// TwinCAT 3 PLC project plc_lfe_vac
// ProgramVersion: 3.1.4022.3
// libraries:
//   L2SI Vacuum Library-TEST, * (SLAC)
//   LCLS General, * (SLAC)
//   PMPS, * (SLAC - LCLS)
//   Tc2_Standard, * (Beckhoff Automation GmbH)
//   Tc2_System, * (Beckhoff Automation GmbH)
//   Tc3_Module, * (Beckhoff Automation GmbH)
// project tree:
//   GVLs/ GVL_Devices.TcGVL, GVL_PMPS.TcGVL (not stored), GVL_PLC_Interfaces.TcGVL (not stored), GVL_Variables.TcGVL
//   / PlcTask.TcTTO (not stored)
//   POUs/ DIAGNOSTICS.TcPOU, MAIN.TcPOU
// real-time tasks:
//   TASK PlcTask: cycle T#10ms, priority 20, ADS port 350
// I/O:
//   DEVICE Device 1 (EtherCAT), AmsNetId 172.21.88.138.2.1
//     PLC_E0_EK1200
// variable links:
//   plc_lfe_vac/plc_lfe_vac Instance <-> Device 1 (EtherCAT)/PLC_E0_EK1200/PLC_E11_EK1122_FEE_Stands/FEE_L0S10_EP1_EP2338-0002
//     PlcTask Inputs/GVL_Devices.MR1L0_HOMS_VGC_01.i_xClsLS <-> Channel 2/Input
//     PlcTask Inputs/GVL_Devices.MR1L0_HOMS_VGC_01.i_xOpnLS <-> Channel 1/Input
//     PlcTask Outputs/GVL_Devices.MR1L0_HOMS_VGC_01.q_xOPN_DO <-> Channel 11/Output
//   plc_lfe_vac/plc_lfe_vac Instance <-> Device 1 (EtherCAT)/PLC_E0_EK1200/PLC_E11_EK1122_FEE_Stands/FEE_L0S14_EP1_EP2338-0002
//     PlcTask Inputs/GVL_Devices.BT2L0_PLEG_VGC_01.i_xClsLS <-> Channel 2/Input
//     PlcTask Inputs/GVL_Devices.BT2L0_PLEG_VGC_01.i_xOpnLS <-> Channel 1/Input
//     PlcTask Outputs/GVL_Devices.BT2L0_PLEG_VGC_01.q_xOPN_DO <-> Channel 11/Output
//   plc_lfe_vac/plc_lfe_vac Instance <-> Device 1 (EtherCAT)/PLC_E0_EK1200/PLC_E11_EK1122_FEE_Stands/FEE_L0S14_EP2_EP3174-0002
//     PlcTask Inputs/GVL_Devices.BT2L0_PLEG_GCC_01.i_iPRESS_R <-> AI Standard Channel 4/Value
//     PlcTask Inputs/GVL_Devices.BT2L0_PLEG_GPI_01.i_iPRESS_R <-> AI Standard Channel 3/Value
//     PlcTask Inputs/GVL_Devices.MR1L1_TXI_GCC_01.i_iPRESS_R <-> AI Standard Channel 2/Value
//     PlcTask Inputs/GVL_Devices.MR1L1_TXI_GPI_01.i_iPRESS_R <-> AI Standard Channel 1/Value
//   plc_lfe_vac/plc_lfe_vac Instance <-> Device 1 (EtherCAT)/PLC_E0_EK1200/PLC_E11_EK1122_FEE_Stands/FEE_L0S14_EP3_EP2624-0002
//     PlcTask Outputs/GVL_Devices.BT2L0_PLEG_GCC_01.q_xHV_DIS <-> Channel 4/Output
//     PlcTask Outputs/GVL_Devices.MR1L1_TXI_GCC_01.q_xHV_DIS <-> Channel 2/Output
//   plc_lfe_vac/plc_lfe_vac Instance <-> Device 1 (EtherCAT)/PLC_E0_EK1200/PLC_E11_EK1122_FEE_Stands/FEE_L0S18_EP1_EP2338-0002
//     PlcTask Inputs/GVL_Devices.MR2L0_HOMS_VGC_01.i_xClsLS <-> Channel 2/Input
//     PlcTask Inputs/GVL_Devices.MR2L0_HOMS_VGC_01.i_xOpnLS <-> Channel 1/Input
//     PlcTask Inputs/GVL_Devices.TV1L1_VGC_01.i_xClsLS <-> Channel 6/Input
//     PlcTask Inputs/GVL_Devices.TV1L1_VGC_01.i_xOpnLS <-> Channel 5/Input
//     PlcTask Outputs/GVL_Devices.MR2L0_HOMS_VGC_01.q_xOPN_DO <-> Channel 11/Output
//     PlcTask Outputs/GVL_Devices.TV1L1_VGC_01.q_xOPN_DO <-> Channel 15/Output
//   plc_lfe_vac/plc_lfe_vac Instance <-> Device 1 (EtherCAT)/PLC_E0_EK1200/PLC_E11_EK1122_FEE_Stands/FEE_L0S18_EP2_EP3174-0002
//     PlcTask Inputs/GVL_Devices.MR2L0_HOMS_GCC_01.i_iPRESS_R <-> AI Standard Channel 2/Value
//     PlcTask Inputs/GVL_Devices.MR2L0_HOMS_GPI_01.i_iPRESS_R <-> AI Standard Channel 1/Value
//   plc_lfe_vac/plc_lfe_vac Instance <-> Device 1 (EtherCAT)/PLC_E0_EK1200/PLC_E11_EK1122_FEE_Stands/FEE_L0S18_EP3_EP2624-0002
//     PlcTask Outputs/GVL_Devices.MR2L0_HOMS_GCC_01.q_xHV_DIS <-> Channel 2/Output
//   plc_lfe_vac/plc_lfe_vac Instance <-> Device 1 (EtherCAT)/PLC_E0_EK1200/PLC_E11_EK1122_FEE_Stands/FEE_L0S19_EP1_EP2338-0002
//     PlcTask Inputs/GVL_Devices.MR2L0_HOMS_VGC_02.i_xClsLS <-> Channel 2/Input
//     PlcTask Inputs/GVL_Devices.MR2L0_HOMS_VGC_02.i_xOpnLS <-> Channel 1/Input
//     PlcTask Inputs/GVL_Devices.PC2L1_L2SI_VGC_01.i_xClsLS <-> Channel 6/Input
//     PlcTask Inputs/GVL_Devices.PC2L1_L2SI_VGC_01.i_xOpnLS <-> Channel 5/Input
//     PlcTask Outputs/GVL_Devices.MR2L0_HOMS_VGC_02.q_xOPN_DO <-> Channel 11/Output
//     PlcTask Outputs/GVL_Devices.PC2L1_L2SI_VGC_01.q_xOPN_DO <-> Channel 15/Output
//   plc_lfe_vac/plc_lfe_vac Instance <-> Device 1 (EtherCAT)/PLC_E0_EK1200/PLC_E11_EK1122_FEE_Stands/FEE_L0S21-2_EP1_EP3174-0002
//     PlcTask Inputs/GVL_Devices.ST1L0_XTES_GCC_01.i_iPRESS_R <-> AI Standard Channel 2/Value
//     PlcTask Inputs/GVL_Devices.ST1L0_XTES_GPI_01.i_iPRESS_R <-> AI Standard Channel 1/Value
//   plc_lfe_vac/plc_lfe_vac Instance <-> Device 1 (EtherCAT)/PLC_E0_EK1200/PLC_E11_EK1122_FEE_Stands/FEE_L0S21-2_EP2_EP2624-0002
//     PlcTask Outputs/GVL_Devices.ST1L0_XTES_GCC_01.q_xHV_DIS <-> Channel 2/Output
//   plc_lfe_vac/plc_lfe_vac Instance <-> Device 1 (EtherCAT)/PLC_E0_EK1200/PLC_E11_EK1122_FEE_Stands/FEE_L0S2_EP1_EP2338-0002
//     PlcTask Inputs/GVL_Devices.TV2L0_VGC_02.i_xClsLS <-> Channel 2/Input
//     PlcTask Inputs/GVL_Devices.TV2L0_VGC_02.i_xOpnLS <-> Channel 1/Input
//     PlcTask Outputs/GVL_Devices.TV2L0_VGC_02.q_xOPN_DO <-> Channel 11/Output
//   plc_lfe_vac/plc_lfe_vac Instance <-> Device 1 (EtherCAT)/PLC_E0_EK1200/PLC_E11_EK1122_FEE_Stands/FEE_L0S8_EP1_EP2338-0002
//     PlcTask Inputs/GVL_Devices.PC1L0_XTES_VGC_01.i_xClsLS <-> Channel 2/Input
//     PlcTask Inputs/GVL_Devices.PC1L0_XTES_VGC_01.i_xOpnLS <-> Channel 1/Input
//     PlcTask Outputs/GVL_Devices.PC1L0_XTES_VGC_01.q_xOPN_DO <-> Channel 11/Output
//   plc_lfe_vac/plc_lfe_vac Instance <-> Device 1 (EtherCAT)/PLC_E0_EK1200/PLC_E12_EK1122_H11_H12/H11_L0S2_EP1_EP2338-0002
//     PlcTask Inputs/GVL_Devices.TV4L0_VGC_01.i_xClsLS <-> Channel 2/Input
//     PlcTask Inputs/GVL_Devices.TV4L0_VGC_01.i_xOpnLS <-> Channel 1/Input
//     PlcTask Outputs/GVL_Devices.TV4L0_VGC_01.q_xOPN_DO <-> Channel 11/Output
//   plc_lfe_vac/plc_lfe_vac Instance <-> Device 1 (EtherCAT)/PLC_E0_EK1200/PLC_E12_EK1122_H11_H12/H11_L0S2_EP2_EP3174-0002
//     PlcTask Inputs/GVL_Devices.TV4L0_GCC_01.i_iPRESS_R <-> AI Standard Channel 2/Value
//     PlcTask Inputs/GVL_Devices.TV4L0_GPI_01.i_iPRESS_R <-> AI Standard Channel 1/Value
//   plc_lfe_vac/plc_lfe_vac Instance <-> Device 1 (EtherCAT)/PLC_E0_EK1200/PLC_E12_EK1122_H11_H12/H11_L0S2_EP3_EP2624-0002
//     PlcTask Outputs/GVL_Devices.TV4L0_GCC_01.q_xHV_DIS <-> Channel 2/Output
//   plc_lfe_vac/plc_lfe_vac Instance <-> Device 1 (EtherCAT)/PLC_E0_EK1200/PLC_E12_EK1122_H11_H12/H11_L0S9_EP1_EP3174-0002
//     PlcTask Inputs/GVL_Devices.TV4L0_GCC_02.i_iPRESS_R <-> AI Standard Channel 2/Value
//     PlcTask Inputs/GVL_Devices.TV4L0_GPI_02.i_iPRESS_R <-> AI Standard Channel 1/Value
//   plc_lfe_vac/plc_lfe_vac Instance <-> Device 1 (EtherCAT)/PLC_E0_EK1200/PLC_E12_EK1122_H11_H12/H11_L0S9_EP2_EP2624-0002
//     PlcTask Outputs/GVL_Devices.TV4L0_GCC_02.q_xHV_DIS <-> Channel 2/Output
//   plc_lfe_vac/plc_lfe_vac Instance <-> Device 1 (EtherCAT)/PLC_E0_EK1200/PLC_E12_EK1122_H11_H12/H12_L0S1_EP1_EP3174-0002
//     PlcTask Inputs/GVL_Devices.TV5L0_GCC_01.i_iPRESS_R <-> AI Standard Channel 2/Value
//     PlcTask Inputs/GVL_Devices.TV5L0_GPI_01.i_iPRESS_R <-> AI Standard Channel 1/Value
//   plc_lfe_vac/plc_lfe_vac Instance <-> Device 1 (EtherCAT)/PLC_E0_EK1200/PLC_E12_EK1122_H11_H12/H12_L0S1_EP2_EP2624-0002
//     PlcTask Outputs/GVL_Devices.TV5L0_GCC_01.q_xHV_DIS <-> Channel 2/Output
//   plc_lfe_vac/plc_lfe_vac Instance <-> Device 1 (EtherCAT)/PLC_E0_EK1200/PLC_E12_EK1122_H11_H12/H12_L0S3_EP1_EP2338-0002
//     PlcTask Inputs/GVL_Devices.TV5L0_VGC_01.i_xClsLS <-> Channel 2/Input
//     PlcTask Inputs/GVL_Devices.TV5L0_VGC_01.i_xOpnLS <-> Channel 1/Input
//     PlcTask Outputs/GVL_Devices.TV5L0_VGC_01.q_xOPN_DO <-> Channel 11/Output
//   plc_lfe_vac/plc_lfe_vac Instance <-> Device 1 (EtherCAT)/PLC_E0_EK1200/PLC_E12_EK1122_H11_H12/H12_L0S3_EP2_EP3174-0002
//     PlcTask Inputs/GVL_Devices.TV5L0_GCC_02.i_iPRESS_R <-> AI Standard Channel 2/Value
//     PlcTask Inputs/GVL_Devices.TV5L0_GCC_03.i_iPRESS_R <-> AI Standard Channel 4/Value
//     PlcTask Inputs/GVL_Devices.TV5L0_GPI_02.i_iPRESS_R <-> AI Standard Channel 1/Value
//   plc_lfe_vac/plc_lfe_vac Instance <-> Device 1 (EtherCAT)/PLC_E0_EK1200/PLC_E12_EK1122_H11_H12/H12_L0S3_EP3_EP2624-0002
//     PlcTask Outputs/GVL_Devices.TV5L0_GCC_02.q_xHV_DIS <-> Channel 2/Output
//     PlcTask Outputs/GVL_Devices.TV5L0_GCC_03.q_xHV_DIS <-> Channel 4/Output
//   plc_lfe_vac/plc_lfe_vac Instance <-> Device 1 (EtherCAT)/PLC_E0_EK1200/PLC_E12_EK1122_H11_H12/H12_L0S6_EP1_EP2338-0002
//     PlcTask Inputs/GVL_Devices.TV6L0_VGC_01.i_xClsLS <-> Channel 2/Input
//     PlcTask Inputs/GVL_Devices.TV6L0_VGC_01.i_xOpnLS <-> Channel 1/Input
//     PlcTask Outputs/GVL_Devices.TV6L0_VGC_01.q_xOPN_DO <-> Channel 11/Output
//   plc_lfe_vac/plc_lfe_vac Instance <-> Device 1 (EtherCAT)/PLC_E0_EK1200/PLC_E1_EL2202
//     PlcTask Outputs/GVL_PMPS.g_FastFaultOutput1.q_xFastFaultOut <-> Channel 1/Output
//     PlcTask Outputs/GVL_PMPS.g_FastFaultOutput2.q_xFastFaultOut <-> Channel 2/Output
//   plc_lfe_vac/plc_lfe_vac Instance <-> Device 1 (EtherCAT)/PLC_E0_EK1200/PLC_E8_EK1122_QpcMks/MKS_E0_EK1100/MKS_E10_EL2794
//     PlcTask Outputs/GVL_Devices.AT2L0_SOLID_GCC_01.q_xHV_DIS <-> Channel 3/Output
//     PlcTask Outputs/GVL_Devices.SL1L0_POWER_GCC_01.q_xHV_DIS <-> Channel 1/Output
//   plc_lfe_vac/plc_lfe_vac Instance <-> Device 1 (EtherCAT)/PLC_E0_EK1200/PLC_E8_EK1122_QpcMks/MKS_E0_EK1100/MKS_E11_EL3064
//     PlcTask Inputs/GVL_Devices.SP1L0_KMONO_GCC_01.i_iPRESS_R <-> AI Standard Channel 1/Value
//   plc_lfe_vac/plc_lfe_vac Instance <-> Device 1 (EtherCAT)/PLC_E0_EK1200/PLC_E8_EK1122_QpcMks/MKS_E0_EK1100/MKS_E12_EL3064
//     PlcTask Inputs/GVL_Devices.SP1L0_KMONO_GPI_01.i_iPRESS_R <-> AI Standard Channel 1/Value
//   plc_lfe_vac/plc_lfe_vac Instance <-> Device 1 (EtherCAT)/PLC_E0_EK1200/PLC_E8_EK1122_QpcMks/MKS_E0_EK1100/MKS_E13_EL2794
//     PlcTask Outputs/GVL_Devices.SP1L0_KMONO_GCC_01.q_xHV_DIS <-> Channel 1/Output
//   plc_lfe_vac/plc_lfe_vac Instance <-> Device 1 (EtherCAT)/PLC_E0_EK1200/PLC_E8_EK1122_QpcMks/MKS_E0_EK1100/MKS_E14_EL3064
//     PlcTask Inputs/GVL_Devices.MR1L0_HOMS_GCC_01.i_iPRESS_R <-> AI Standard Channel 3/Value
//     PlcTask Inputs/GVL_Devices.PA1L0_GCC_01.i_iPRESS_R <-> AI Standard Channel 1/Value
//   plc_lfe_vac/plc_lfe_vac Instance <-> Device 1 (EtherCAT)/PLC_E0_EK1200/PLC_E8_EK1122_QpcMks/MKS_E0_EK1100/MKS_E15_EL3064
//     PlcTask Inputs/GVL_Devices.MR1L0_HOMS_GPI_01.i_iPRESS_R <-> AI Standard Channel 2/Value
//     PlcTask Inputs/GVL_Devices.PA1L0_GPI_01.i_iPRESS_R <-> AI Standard Channel 1/Value
//   plc_lfe_vac/plc_lfe_vac Instance <-> Device 1 (EtherCAT)/PLC_E0_EK1200/PLC_E8_EK1122_QpcMks/MKS_E0_EK1100/MKS_E16_EL2794
//     PlcTask Outputs/GVL_Devices.MR1L0_HOMS_GCC_01.q_xHV_DIS <-> Channel 3/Output
//     PlcTask Outputs/GVL_Devices.PA1L0_GCC_01.q_xHV_DIS <-> Channel 1/Output
//   plc_lfe_vac/plc_lfe_vac Instance <-> Device 1 (EtherCAT)/PLC_E0_EK1200/PLC_E8_EK1122_QpcMks/MKS_E0_EK1100/MKS_E18_EL3064
//     PlcTask Inputs/GVL_Devices.TV2L0_GFS_01.i_iPRESS_R <-> AI Standard Channel 1/Value
//     PlcTask Inputs/GVL_Devices.TV5L0_GFS_01.i_iPRESS_R <-> AI Standard Channel 3/Value
//   plc_lfe_vac/plc_lfe_vac Instance <-> Device 1 (EtherCAT)/PLC_E0_EK1200/PLC_E8_EK1122_QpcMks/MKS_E0_EK1100/MKS_E1_EL3064
//     PlcTask Inputs/GVL_Devices.TV1L0_GCC_01.i_iPRESS_R <-> AI Standard Channel 1/Value
//     PlcTask Inputs/GVL_Devices.TV2L0_GCC_01.i_iPRESS_R <-> AI Standard Channel 3/Value
//   plc_lfe_vac/plc_lfe_vac Instance <-> Device 1 (EtherCAT)/PLC_E0_EK1200/PLC_E8_EK1122_QpcMks/MKS_E0_EK1100/MKS_E20_EL2794
//     PlcTask Outputs/GVL_Devices.TV2L0_GFS_01.q_xHV_DIS <-> Channel 1/Output
//     PlcTask Outputs/GVL_Devices.TV5L0_GFS_01.q_xHV_DIS <-> Channel 2/Output
//   plc_lfe_vac/plc_lfe_vac Instance <-> Device 1 (EtherCAT)/PLC_E0_EK1200/PLC_E8_EK1122_QpcMks/MKS_E0_EK1100/MKS_E2_EL3064
//     PlcTask Inputs/GVL_Devices.TV1L0_GPI_01.i_iPRESS_R <-> AI Standard Channel 1/Value
//     PlcTask Inputs/GVL_Devices.TV2L0_GPI_01.i_iPRESS_R <-> AI Standard Channel 2/Value
//   plc_lfe_vac/plc_lfe_vac Instance <-> Device 1 (EtherCAT)/PLC_E0_EK1200/PLC_E8_EK1122_QpcMks/MKS_E0_EK1100/MKS_E3_EL2794
//     PlcTask Outputs/GVL_Devices.TV1L0_GCC_01.q_xHV_DIS <-> Channel 1/Output
//     PlcTask Outputs/GVL_Devices.TV2L0_GCC_01.q_xHV_DIS <-> Channel 3/Output
//   plc_lfe_vac/plc_lfe_vac Instance <-> Device 1 (EtherCAT)/PLC_E0_EK1200/PLC_E8_EK1122_QpcMks/MKS_E0_EK1100/MKS_E4_EL3064
//     PlcTask Inputs/GVL_Devices.TV2L0_GCC_02.i_iPRESS_R <-> AI Standard Channel 1/Value
//   plc_lfe_vac/plc_lfe_vac Instance <-> Device 1 (EtherCAT)/PLC_E0_EK1200/PLC_E8_EK1122_QpcMks/MKS_E0_EK1100/MKS_E5_EL3064
//     PlcTask Inputs/GVL_Devices.TV2L0_GPI_02.i_iPRESS_R <-> AI Standard Channel 1/Value
//   plc_lfe_vac/plc_lfe_vac Instance <-> Device 1 (EtherCAT)/PLC_E0_EK1200/PLC_E8_EK1122_QpcMks/MKS_E0_EK1100/MKS_E6_EL2794
//     PlcTask Outputs/GVL_Devices.TV2L0_GCC_02.q_xHV_DIS <-> Channel 1/Output
//   plc_lfe_vac/plc_lfe_vac Instance <-> Device 1 (EtherCAT)/PLC_E0_EK1200/PLC_E8_EK1122_QpcMks/MKS_E0_EK1100/MKS_E8_EL3064
//     PlcTask Inputs/GVL_Devices.AT2L0_SOLID_GCC_01.i_iPRESS_R <-> AI Standard Channel 3/Value
//     PlcTask Inputs/GVL_Devices.SL1L0_POWER_GCC_01.i_iPRESS_R <-> AI Standard Channel 1/Value
//   plc_lfe_vac/plc_lfe_vac Instance <-> Device 1 (EtherCAT)/PLC_E0_EK1200/PLC_E8_EK1122_QpcMks/MKS_E0_EK1100/MKS_E9_EL3064
//     PlcTask Inputs/GVL_Devices.AT2L0_SOLID_GPI_01.i_iPRESS_R <-> AI Standard Channel 2/Value
//     PlcTask Inputs/GVL_Devices.SL1L0_POWER_GPI_01.i_iPRESS_R <-> AI Standard Channel 1/Value
//   plc_lfe_vac/plc_lfe_vac Instance <-> Device 1 (EtherCAT)/PLC_E0_EK1200/PLC_E8_EK1122_QpcMks/QPC_E0_EK1100/QPC_E11_EL3064
//     PlcTask Inputs/GVL_Devices.BT2L0_PLEG_PIP_01.i_iPRESS <-> AI Standard Channel 3/Value
//     PlcTask Inputs/GVL_Devices.MR2L0_HOMS_PIP_01.i_iPRESS <-> AI Standard Channel 4/Value
//     PlcTask Inputs/GVL_Devices.SP1L0_KMONO_PIP_01.i_iPRESS <-> AI Standard Channel 1/Value
//   plc_lfe_vac/plc_lfe_vac Instance <-> Device 1 (EtherCAT)/PLC_E0_EK1200/PLC_E8_EK1122_QpcMks/QPC_E0_EK1100/QPC_E12_EL1004
//     PlcTask Inputs/GVL_Devices.BT2L0_PLEG_PIP_01.i_xSP_DI <-> Channel 3/Input
//     PlcTask Inputs/GVL_Devices.MR2L0_HOMS_PIP_01.i_xSP_DI <-> Channel 4/Input
//     PlcTask Inputs/GVL_Devices.SP1L0_KMONO_PIP_01.i_xSP_DI <-> Channel 1/Input
//   plc_lfe_vac/plc_lfe_vac Instance <-> Device 1 (EtherCAT)/PLC_E0_EK1200/PLC_E8_EK1122_QpcMks/QPC_E0_EK1100/QPC_E13_EL2794
//     PlcTask Outputs/GVL_Devices.BT2L0_PLEG_PIP_01.q_xHVEna_DO <-> Channel 3/Output
//     PlcTask Outputs/GVL_Devices.MR2L0_HOMS_PIP_01.q_xHVEna_DO <-> Channel 4/Output
//     PlcTask Outputs/GVL_Devices.SP1L0_KMONO_PIP_01.q_xHVEna_DO <-> Channel 1/Output
//   plc_lfe_vac/plc_lfe_vac Instance <-> Device 1 (EtherCAT)/PLC_E0_EK1200/PLC_E8_EK1122_QpcMks/QPC_E0_EK1100/QPC_E14_EL3064
//     PlcTask Inputs/GVL_Devices.MR1L0_HOMS_PIP_01.i_iPRESS <-> AI Standard Channel 4/Value
//     PlcTask Inputs/GVL_Devices.MR1L1_TXI_PIP_01.i_iPRESS <-> AI Standard Channel 3/Value
//     PlcTask Inputs/GVL_Devices.ST1L0_XTES_PIP_01.i_iPRESS <-> AI Standard Channel 2/Value
//     PlcTask Inputs/GVL_Devices.TV3L0_PIP_01.i_iPRESS <-> AI Standard Channel 1/Value
//   plc_lfe_vac/plc_lfe_vac Instance <-> Device 1 (EtherCAT)/PLC_E0_EK1200/PLC_E8_EK1122_QpcMks/QPC_E0_EK1100/QPC_E15_EL1004
//     PlcTask Inputs/GVL_Devices.MR1L0_HOMS_PIP_01.i_xSP_DI <-> Channel 4/Input
//     PlcTask Inputs/GVL_Devices.MR1L1_TXI_PIP_01.i_xSP_DI <-> Channel 3/Input
//     PlcTask Inputs/GVL_Devices.ST1L0_XTES_PIP_01.i_xSP_DI <-> Channel 2/Input
//     PlcTask Inputs/GVL_Devices.TV3L0_PIP_01.i_xSP_DI <-> Channel 1/Input
//   plc_lfe_vac/plc_lfe_vac Instance <-> Device 1 (EtherCAT)/PLC_E0_EK1200/PLC_E8_EK1122_QpcMks/QPC_E0_EK1100/QPC_E16_EL2794
//     PlcTask Outputs/GVL_Devices.MR1L0_HOMS_PIP_01.q_xHVEna_DO <-> Channel 4/Output
//     PlcTask Outputs/GVL_Devices.MR1L1_TXI_PIP_01.q_xHVEna_DO <-> Channel 3/Output
//     PlcTask Outputs/GVL_Devices.ST1L0_XTES_PIP_01.q_xHVEna_DO <-> Channel 2/Output
//     PlcTask Outputs/GVL_Devices.TV3L0_PIP_01.q_xHVEna_DO <-> Channel 1/Output
//   plc_lfe_vac/plc_lfe_vac Instance <-> Device 1 (EtherCAT)/PLC_E0_EK1200/PLC_E8_EK1122_QpcMks/QPC_E0_EK1100/QPC_E17_EL3064
//     PlcTask Inputs/GVL_Devices.TV4L0_PIP_01.i_iPRESS <-> AI Standard Channel 1/Value
//     PlcTask Inputs/GVL_Devices.TV4L0_PIP_02.i_iPRESS <-> AI Standard Channel 2/Value
//     PlcTask Inputs/GVL_Devices.TV5L0_PIP_01.i_iPRESS <-> AI Standard Channel 3/Value
//     PlcTask Inputs/GVL_Devices.TV5L0_PIP_02.i_iPRESS <-> AI Standard Channel 4/Value
//   plc_lfe_vac/plc_lfe_vac Instance <-> Device 1 (EtherCAT)/PLC_E0_EK1200/PLC_E8_EK1122_QpcMks/QPC_E0_EK1100/QPC_E18_EL1004
//     PlcTask Inputs/GVL_Devices.TV4L0_PIP_01.i_xSP_DI <-> Channel 1/Input
//     PlcTask Inputs/GVL_Devices.TV4L0_PIP_02.i_xSP_DI <-> Channel 2/Input
//     PlcTask Inputs/GVL_Devices.TV5L0_PIP_01.i_xSP_DI <-> Channel 3/Input
//     PlcTask Inputs/GVL_Devices.TV5L0_PIP_02.i_xSP_DI <-> Channel 4/Input
//   plc_lfe_vac/plc_lfe_vac Instance <-> Device 1 (EtherCAT)/PLC_E0_EK1200/PLC_E8_EK1122_QpcMks/QPC_E0_EK1100/QPC_E19_EL2794
//     PlcTask Outputs/GVL_Devices.TV4L0_PIP_01.q_xHVEna_DO <-> Channel 1/Output
//     PlcTask Outputs/GVL_Devices.TV4L0_PIP_02.q_xHVEna_DO <-> Channel 2/Output
//     PlcTask Outputs/GVL_Devices.TV5L0_PIP_01.q_xHVEna_DO <-> Channel 3/Output
//     PlcTask Outputs/GVL_Devices.TV5L0_PIP_02.q_xHVEna_DO <-> Channel 4/Output
//   plc_lfe_vac/plc_lfe_vac Instance <-> Device 1 (EtherCAT)/PLC_E0_EK1200/PLC_E8_EK1122_QpcMks/QPC_E0_EK1100/QPC_E1_EL3064
//     PlcTask Inputs/GVL_Devices.RTDSL0_PIP_01.i_iPRESS <-> AI Standard Channel 1/Value
//     PlcTask Inputs/GVL_Devices.RTDSL0_PIP_02.i_iPRESS <-> AI Standard Channel 2/Value
//     PlcTask Inputs/GVL_Devices.RTDSL0_PIP_03.i_iPRESS <-> AI Standard Channel 3/Value
//     PlcTask Inputs/GVL_Devices.RTDSL0_PIP_04.i_iPRESS <-> AI Standard Channel 4/Value
//   plc_lfe_vac/plc_lfe_vac Instance <-> Device 1 (EtherCAT)/PLC_E0_EK1200/PLC_E8_EK1122_QpcMks/QPC_E0_EK1100/QPC_E21_EL3064
//     PlcTask Inputs/GVL_Devices.AT2L0_SOLID_PIN_01.i_iPRESS <-> AI Standard Channel 2/Value
//     PlcTask Inputs/GVL_Devices.PA1L0_PIN_01.i_iPRESS <-> AI Standard Channel 3/Value
//     PlcTask Inputs/GVL_Devices.PA2L0_PIN_01.i_iPRESS <-> AI Standard Channel 4/Value
//     PlcTask Inputs/GVL_Devices.SL1L0_POWER_PIN_01.i_iPRESS <-> AI Standard Channel 1/Value
//   plc_lfe_vac/plc_lfe_vac Instance <-> Device 1 (EtherCAT)/PLC_E0_EK1200/PLC_E8_EK1122_QpcMks/QPC_E0_EK1100/QPC_E22_EL1004
//     PlcTask Inputs/GVL_Devices.AT2L0_SOLID_PIN_01.i_xSP_DI <-> Channel 2/Input
//     PlcTask Inputs/GVL_Devices.PA1L0_PIN_01.i_xSP_DI <-> Channel 3/Input
//     PlcTask Inputs/GVL_Devices.PA2L0_PIN_01.i_xSP_DI <-> Channel 4/Input
//     PlcTask Inputs/GVL_Devices.SL1L0_POWER_PIN_01.i_xSP_DI <-> Channel 1/Input
//   plc_lfe_vac/plc_lfe_vac Instance <-> Device 1 (EtherCAT)/PLC_E0_EK1200/PLC_E8_EK1122_QpcMks/QPC_E0_EK1100/QPC_E23_EL2794
//     PlcTask Outputs/GVL_Devices.AT2L0_SOLID_PIN_01.q_xHVEna_DO <-> Channel 2/Output
//     PlcTask Outputs/GVL_Devices.PA1L0_PIN_01.q_xHVEna_DO <-> Channel 3/Output
//     PlcTask Outputs/GVL_Devices.PA2L0_PIN_01.q_xHVEna_DO <-> Channel 4/Output
//     PlcTask Outputs/GVL_Devices.SL1L0_POWER_PIN_01.q_xHVEna_DO <-> Channel 1/Output
//   plc_lfe_vac/plc_lfe_vac Instance <-> Device 1 (EtherCAT)/PLC_E0_EK1200/PLC_E8_EK1122_QpcMks/QPC_E0_EK1100/QPC_E2_EL1004
//     PlcTask Inputs/GVL_Devices.RTDSL0_PIP_01.i_xSP_DI <-> Channel 1/Input
//     PlcTask Inputs/GVL_Devices.RTDSL0_PIP_02.i_xSP_DI <-> Channel 2/Input
//     PlcTask Inputs/GVL_Devices.RTDSL0_PIP_03.i_xSP_DI <-> Channel 3/Input
//     PlcTask Inputs/GVL_Devices.RTDSL0_PIP_04.i_xSP_DI <-> Channel 4/Input
//   plc_lfe_vac/plc_lfe_vac Instance <-> Device 1 (EtherCAT)/PLC_E0_EK1200/PLC_E8_EK1122_QpcMks/QPC_E0_EK1100/QPC_E3_EL2794
//     PlcTask Outputs/GVL_Devices.RTDSL0_PIP_01.q_xHVEna_DO <-> Channel 1/Output
//     PlcTask Outputs/GVL_Devices.RTDSL0_PIP_02.q_xHVEna_DO <-> Channel 2/Output
//     PlcTask Outputs/GVL_Devices.RTDSL0_PIP_03.q_xHVEna_DO <-> Channel 3/Output
//     PlcTask Outputs/GVL_Devices.RTDSL0_PIP_04.q_xHVEna_DO <-> Channel 4/Output
//   plc_lfe_vac/plc_lfe_vac Instance <-> Device 1 (EtherCAT)/PLC_E0_EK1200/PLC_E8_EK1122_QpcMks/QPC_E0_EK1100/QPC_E4_EL3064
//     PlcTask Inputs/GVL_Devices.IM1L0_XTES_PIP_01.i_iPRESS <-> AI Standard Channel 2/Value
//     PlcTask Inputs/GVL_Devices.RTDSL0_PIP_05.i_iPRESS <-> AI Standard Channel 1/Value
//     PlcTask Inputs/GVL_Devices.TV5L0_PIP_03.i_iPRESS <-> AI Standard Channel 4/Value
//   plc_lfe_vac/plc_lfe_vac Instance <-> Device 1 (EtherCAT)/PLC_E0_EK1200/PLC_E8_EK1122_QpcMks/QPC_E0_EK1100/QPC_E5_EL1004
//     PlcTask Inputs/GVL_Devices.IM1L0_XTES_PIP_01.i_xSP_DI <-> Channel 2/Input
//     PlcTask Inputs/GVL_Devices.RTDSL0_PIP_05.i_xSP_DI <-> Channel 1/Input
//     PlcTask Inputs/GVL_Devices.TV5L0_PIP_03.i_xSP_DI <-> Channel 4/Input
//   plc_lfe_vac/plc_lfe_vac Instance <-> Device 1 (EtherCAT)/PLC_E0_EK1200/PLC_E8_EK1122_QpcMks/QPC_E0_EK1100/QPC_E6_EL2794
//     PlcTask Outputs/GVL_Devices.IM1L0_XTES_PIP_01.q_xHVEna_DO <-> Channel 2/Output
//     PlcTask Outputs/GVL_Devices.RTDSL0_PIP_05.q_xHVEna_DO <-> Channel 1/Output
//     PlcTask Outputs/GVL_Devices.TV5L0_PIP_03.q_xHVEna_DO <-> Channel 4/Output
//   plc_lfe_vac/plc_lfe_vac Instance <-> Device 1 (EtherCAT)/PLC_E0_EK1200/PLC_E8_EK1122_QpcMks/QPC_E0_EK1100/QPC_E7_EL3064
//     PlcTask Inputs/GVL_Devices.TV2L0_PIP_01.i_iPRESS <-> AI Standard Channel 1/Value
//     PlcTask Inputs/GVL_Devices.TV2L0_PIP_02.i_iPRESS <-> AI Standard Channel 2/Value
//     PlcTask Inputs/GVL_Devices.TV2L0_PIP_03.i_iPRESS <-> AI Standard Channel 3/Value
//   plc_lfe_vac/plc_lfe_vac Instance <-> Device 1 (EtherCAT)/PLC_E0_EK1200/PLC_E8_EK1122_QpcMks/QPC_E0_EK1100/QPC_E8_EL1004
//     PlcTask Inputs/GVL_Devices.TV2L0_PIP_01.i_xSP_DI <-> Channel 1/Input
//     PlcTask Inputs/GVL_Devices.TV2L0_PIP_02.i_xSP_DI <-> Channel 2/Input
//     PlcTask Inputs/GVL_Devices.TV2L0_PIP_03.i_xSP_DI <-> Channel 3/Input
//   plc_lfe_vac/plc_lfe_vac Instance <-> Device 1 (EtherCAT)/PLC_E0_EK1200/PLC_E8_EK1122_QpcMks/QPC_E0_EK1100/QPC_E9_EL2794
//     PlcTask Outputs/GVL_Devices.TV2L0_PIP_01.q_xHVEna_DO <-> Channel 1/Output
//     PlcTask Outputs/GVL_Devices.TV2L0_PIP_02.q_xHVEna_DO <-> Channel 2/Output
//     PlcTask Outputs/GVL_Devices.TV2L0_PIP_03.q_xHVEna_DO <-> Channel 3/Output
//   plc_lfe_vac/plc_lfe_vac Instance <-> Device 1 (EtherCAT)/PLC_E0_EK1200/PLC_E9_EK1122_EBD/EBD_E0_EK1100/EBD_E1_EL1004
//     PlcTask Inputs/GVL_Devices.IM1L0_XTES_VGC_01.i_xClsLS <-> Channel 4/Input
//     PlcTask Inputs/GVL_Devices.IM1L0_XTES_VGC_01.i_xOpnLS <-> Channel 3/Input
//     PlcTask Inputs/GVL_Devices.TV1L0_VGC_01.i_xClsLS <-> Channel 2/Input
//     PlcTask Inputs/GVL_Devices.TV1L0_VGC_01.i_xOpnLS <-> Channel 1/Input
//   plc_lfe_vac/plc_lfe_vac Instance <-> Device 1 (EtherCAT)/PLC_E0_EK1200/PLC_E9_EK1122_EBD/EBD_E0_EK1100/EBD_E2_EL2004
//     PlcTask Outputs/GVL_Devices.IM1L0_XTES_VGC_01.q_xOPN_DO <-> Channel 3/Output
//     PlcTask Outputs/GVL_Devices.IM1L0_XTES_VGC_01.q_xOPN_DO_2 <-> Channel 4/Output
//     PlcTask Outputs/GVL_Devices.TV1L0_VGC_01.q_xOPN_DO <-> Channel 1/Output
//     PlcTask Outputs/GVL_Devices.TV1L0_VGC_01.q_xOPN_DO_2 <-> Channel 2/Output
//   plc_lfe_vac/plc_lfe_vac Instance <-> Device 1 (EtherCAT)/PLC_E0_EK1200/PLC_E9_EK1122_EBD/EBD_E0_EK1100/EBD_E3_EL1004
//     PlcTask Inputs/GVL_Devices.TV2L0_VGC_01.i_xClsLS <-> Channel 2/Input
//     PlcTask Inputs/GVL_Devices.TV2L0_VGC_01.i_xOpnLS <-> Channel 1/Input
//   plc_lfe_vac/plc_lfe_vac Instance <-> Device 1 (EtherCAT)/PLC_E0_EK1200/PLC_E9_EK1122_EBD/EBD_E0_EK1100/EBD_E4_EL2004
//     PlcTask Outputs/GVL_Devices.TV2L0_VGC_01.q_xOPN_DO <-> Channel 1/Output
//     PlcTask Outputs/GVL_Devices.TV2L0_VGC_01.q_xOPN_DO_2 <-> Channel 2/Output
//   plc_lfe_vac/plc_lfe_vac Instance <-> Device 1 (EtherCAT)/PLC_E0_EK1200/PLC_E9_EK1122_EBD/EBD_E0_EK1100/EBD_E5_EL1008
//     PlcTask Inputs/MAIN.i_xUpstreamTreaty_PressOK <-> Channel 1/Input
//   plc_lfe_vac/plc_lfe_vac Instance <-> plc_lfe_vac_fs/plc_lfe_vac_fs Instance
//     PlcTask Inputs/GVL_Devices.PA1L0_VFS_01.i_xTrigger <-> PlcTask Outputs/GVL_FS_Devices.PA1L0_VFS_01.q_xTrigger
//     PlcTask Inputs/GVL_Devices.PA1L0_VFS_01.i_xVAC_FAULT_OK <-> PlcTask Outputs/GVL_FS_Devices.PA1L0_VFS_01.q_xVAC_FAULT_OK
//     PlcTask Inputs/GVL_Devices.PA1L0_VFS_01.i_xVFS_Closed <-> PlcTask Outputs/GVL_FS_Devices.PA1L0_VFS_01.q_xVFS_Closed
//     PlcTask Inputs/GVL_Devices.PA1L0_VFS_01.i_xVFS_Open <-> PlcTask Outputs/GVL_FS_Devices.PA1L0_VFS_01.q_xVFS_Open
//     PlcTask Inputs/GVL_Devices.TV3L0_VFS_01_Interface.i_xTrigger <-> PlcTask Outputs/GVL_FS_Devices.TV3L0_VFS_01.q_xTrigger
//     PlcTask Inputs/GVL_Devices.TV3L0_VFS_01_Interface.i_xVAC_FAULT_OK <-> PlcTask Outputs/GVL_FS_Devices.TV3L0_VFS_01.q_xVAC_FAULT_OK
//     PlcTask Inputs/GVL_Devices.TV3L0_VFS_01_Interface.i_xVFS_Closed <-> PlcTask Outputs/GVL_FS_Devices.TV3L0_VFS_01.q_xVFS_Closed
//     PlcTask Inputs/GVL_Devices.TV3L0_VFS_01_Interface.i_xVFS_Open <-> PlcTask Outputs/GVL_FS_Devices.TV3L0_VFS_01.q_xVFS_Open
//     PlcTask Outputs/GVL_Devices.PA1L0_VFS_01.q_xPRESS_OK <-> PlcTask Inputs/GVL_FS_Devices.PA1L0_VFS_01.i_xPress_OK
//     PlcTask Outputs/GVL_Devices.PA1L0_VFS_01.q_xVAC_FAULT_Reset <-> PlcTask Inputs/GVL_FS_Devices.PA1L0_VFS_01.i_xResetFault
//     PlcTask Outputs/GVL_Devices.TV3L0_VFS_01_Interface.q_xPRESS_OK <-> PlcTask Inputs/GVL_FS_Devices.TV3L0_VFS_01.i_xPress_OK
//     PlcTask Outputs/GVL_Devices.TV3L0_VFS_01_Interface.q_xVAC_FAULT_Reset <-> PlcTask Inputs/GVL_FS_Devices.TV3L0_VFS_01.i_xResetFault
//   plc_lfe_vac_fs Instance <-> Device 1 (EtherCAT)/PLC_E0_EK1200/PLC_E7_EK1122_QpcMks/MKS_E0_EK1100/MKS_E22_EL1124
//     PlcTask Inputs/GVL_FS_Devices.PA1L0_VFS_01.i_xTrigger <-> Channel 1/Input
//     PlcTask Inputs/GVL_FS_Devices.TV3L0_VFS_01.i_xTrigger <-> Channel 2/Input
//   plc_lfe_vac_fs Instance <-> Device 1 (EtherCAT)/PLC_E0_EK1200/PLC_E9_EK1122_FSV/FSV1_E0_EK1100_L0S10/FSV1_E1_EL1004
//     PlcTask Inputs/GVL_FS_Devices.PA1L0_VFS_01.i_xClsLS <-> Channel 1/Input
//     PlcTask Inputs/GVL_FS_Devices.PA1L0_VFS_01.i_xOpnLS <-> Channel 2/Input
//   plc_lfe_vac_fs Instance <-> Device 1 (EtherCAT)/PLC_E0_EK1200/PLC_E9_EK1122_FSV/FSV1_E0_EK1100_L0S10/FSV1_E3_EL2212
//     PlcTask Outputs/GVL_FS_Devices.PA1L0_VFS_01.q_xClose_A <-> DOX Control Channel 1/Control/Output
//     PlcTask Outputs/GVL_FS_Devices.PA1L0_VFS_01.q_xClose_B <-> DOX Control Channel 2/Control/Output
//   plc_lfe_vac_fs Instance <-> Device 1 (EtherCAT)/PLC_E0_EK1200/PLC_E9_EK1122_FSV/FSV1_E0_EK1100_L0S10/FSV1_E4_EL2212
//     PlcTask Outputs/GVL_FS_Devices.PA1L0_VFS_01.q_xClose_C <-> DOX Control Channel 1/Control/Output
//     PlcTask Outputs/GVL_FS_Devices.PA1L0_VFS_01.q_xOPN_DO <-> DOX Control Channel 2/Control/Output
//   plc_lfe_vac_fs Instance <-> Device 1 (EtherCAT)/PLC_E0_EK1200/PLC_E9_EK1122_FSV/FSV2_E0_EK1100_L0S19/FSV2_E1_EL1004
//     PlcTask Inputs/GVL_FS_Devices.TV3L0_VFS_01.i_xClsLS <-> Channel 1/Input
//     PlcTask Inputs/GVL_FS_Devices.TV3L0_VFS_01.i_xOpnLS <-> Channel 2/Input
//   plc_lfe_vac_fs Instance <-> Device 1 (EtherCAT)/PLC_E0_EK1200/PLC_E9_EK1122_FSV/FSV2_E0_EK1100_L0S19/FSV2_E3_EL2212
//     PlcTask Outputs/GVL_FS_Devices.TV3L0_VFS_01.q_xClose_A <-> DOX Control Channel 1/Control/Output
//     PlcTask Outputs/GVL_FS_Devices.TV3L0_VFS_01.q_xClose_B <-> DOX Control Channel 2/Control/Output
//   plc_lfe_vac_fs Instance <-> Device 1 (EtherCAT)/PLC_E0_EK1200/PLC_E9_EK1122_FSV/FSV2_E0_EK1100_L0S19/FSV2_E4_EL2212
//     PlcTask Outputs/GVL_FS_Devices.TV3L0_VFS_01.q_xClose_C <-> DOX Control Channel 1/Control/Output
//     PlcTask Outputs/GVL_FS_Devices.TV3L0_VFS_01.q_xOPN_DO <-> DOX Control Channel 2/Control/Output

// ---- GVLs/GVL_Devices.TcGVL
//{attribute 'qualified_only'}
VAR_GLOBAL
	

(*TRANSPORT VACUUM 1 HXR 0 LINE*) //HXR INSTALLATION SECTION 1
	{attribute 'TcLinkTo' := 	'.i_xOpnLS	:=	TIIB[EBD_E1_EL1004]^Channel 1^Input;
								 .i_xClsLS	:=	TIIB[EBD_E1_EL1004]^Channel 2^Input;
								 .q_xOPN_DO	:=	TIIB[EBD_E2_EL2004]^Channel 1^Output;
								 .q_xOPN_DO_2	:=	TIIB[EBD_E2_EL2004]^Channel 2^Output
	'}
	{attribute 'pytmc' := '
		pv: TV1L0:VGC:01
		io: io
	'}
	TV1L0_VGC_01 : FB_VGC_EBD;
	
	{attribute 'TcLinkTo' := 	'.i_iPRESS_R	:=	TIIB[MKS_E2_EL3064]^AI Standard Channel 1^Value
	'}
	{attribute 'pytmc' := '
		pv: TV1L0:GPI:01
		io: io
	'}
	TV1L0_GPI_01 : FB_MKS317;
	
	{attribute 'TcLinkTo' := 	'.i_iPRESS_R	:=	TIIB[MKS_E1_EL3064]^AI Standard Channel 1^Value;
								 .q_xHV_DIS		:= 	TIIB[MKS_E3_EL2794]^Channel 1^Output
	'}
	{attribute 'pytmc' := '
		pv: TV1L0:GCC:01
		io: io
	'}
	TV1L0_GCC_01 : FB_MKS422;
	
(*RAPID TRANSIT DIAGNOSTIC STAND HXR 0 LINE*)
	{attribute 'TcLinkTo' := 	'.i_iPRESS		:=	TIIB[QPC_E1_EL3064]^AI Standard Channel 1^Value;
								 .i_xSP_DI		:= 	TIIB[QPC_E2_EL1004]^Channel 1^Input;
								 .q_xHVEna_DO	:= 	TIIB[QPC_E3_EL2794]^Channel 1^Output
	'}
	{attribute 'pytmc' := '
		pv: RTDSL0:PIP:01
		io: io
	'}
	RTDSL0_PIP_01 : FB_PIP_Gamma;

	{attribute 'TcLinkTo' := 	'.i_iPRESS		:=	TIIB[QPC_E1_EL3064]^AI Standard Channel 2^Value;
								 .i_xSP_DI		:= 	TIIB[QPC_E2_EL1004]^Channel 2^Input;
								 .q_xHVEna_DO	:= 	TIIB[QPC_E3_EL2794]^Channel 2^Output
	'}	
	{attribute 'pytmc' := '
		pv: RTDSL0:PIP:02
		io: io
	'}
	RTDSL0_PIP_02 : FB_PIP_Gamma;
	
	{attribute 'TcLinkTo' := 	'.i_iPRESS		:=	TIIB[QPC_E1_EL3064]^AI Standard Channel 3^Value;
								 .i_xSP_DI		:= 	TIIB[QPC_E2_EL1004]^Channel 3^Input;
								 .q_xHVEna_DO	:= 	TIIB[QPC_E3_EL2794]^Channel 3^Output
	'}
	{attribute 'pytmc' := '
		pv: RTDSL0:PIP:03
		io: io
	'}
	RTDSL0_PIP_03 : FB_PIP_Gamma;

	{attribute 'TcLinkTo' := 	'.i_iPRESS		:=	TIIB[QPC_E1_EL3064]^AI Standard Channel 4^Value;
								 .i_xSP_DI		:= 	TIIB[QPC_E2_EL1004]^Channel 4^Input;
								 .q_xHVEna_DO	:= 	TIIB[QPC_E3_EL2794]^Channel 4^Output
	'}	
	{attribute 'pytmc' := '
		pv: RTDSL0:PIP:04
		io: io
	'}
	RTDSL0_PIP_04 : FB_PIP_Gamma;

	{attribute 'TcLinkTo' := 	'.i_iPRESS		:=	TIIB[QPC_E4_EL3064]^AI Standard Channel 1^Value;
								 .i_xSP_DI		:= 	TIIB[QPC_E5_EL1004]^Channel 1^Input;
								 .q_xHVEna_DO	:= 	TIIB[QPC_E6_EL2794]^Channel 1^Output
	'}	
	{attribute 'pytmc' := '
		pv: RTDSL0:PIP:05
		io: io
	'}
	RTDSL0_PIP_05 : FB_PIP_Gamma;

(* IM1L0-XTES*) //HXR INSTALLATION SECTION 2
	{attribute 'TcLinkTo' := 	'.i_xOpnLS	:=	TIIB[EBD_E1_EL1004]^Channel 3^Input;
								 .i_xClsLS	:=	TIIB[EBD_E1_EL1004]^Channel 4^Input;
								 .q_xOPN_DO	:=	TIIB[EBD_E2_EL2004]^Channel 3^Output;
								 .q_xOPN_DO_2	:=	TIIB[EBD_E2_EL2004]^Channel 4^Output
	'}
	{attribute 'pytmc' := '
		pv: IM1L0:XTES:VGC:01
		io: io
	'}
	IM1L0_XTES_VGC_01 : FB_VGC_EBD;

	{attribute 'TcLinkTo' := 	'.i_iPRESS		:=	TIIB[QPC_E4_EL3064]^AI Standard Channel 2^Value;
								 .i_xSP_DI		:= 	TIIB[QPC_E5_EL1004]^Channel 2^Input;
								 .q_xHVEna_DO	:= 	TIIB[QPC_E6_EL2794]^Channel 2^Output
	'}	
	{attribute 'pytmc' := '
		pv: IM1L0:XTES:PIP:01
		io: io
	'}
	IM1L0_XTES_PIP_01 : FB_PIP_Gamma;
	
(*TV2L0*)
	{attribute 'TcLinkTo' := 	'.i_iPRESS		:=	TIIB[QPC_E7_EL3064]^AI Standard Channel 1^Value;
								 .i_xSP_DI		:= 	TIIB[QPC_E8_EL1004]^Channel 1^Input;
								 .q_xHVEna_DO	:= 	TIIB[QPC_E9_EL2794]^Channel 1^Output
	'}
	{attribute 'pytmc' := '
		pv: TV2L0:PIP:01
		io: io
	'}
	TV2L0_PIP_01 : FB_PIP_Gamma;
	
	{attribute 'TcLinkTo' := 	'.i_iPRESS_R	:=	TIIB[MKS_E2_EL3064]^AI Standard Channel 2^Value
	'}
	{attribute 'pytmc' := '
		pv: TV2L0:GPI:01
		io: io
	'}
	TV2L0_GPI_01 : FB_MKS317;

	{attribute 'TcLinkTo' := 	'.i_iPRESS_R	:=	TIIB[MKS_E1_EL3064]^AI Standard Channel 3^Value;
								 .q_xHV_DIS		:= 	TIIB[MKS_E3_EL2794]^Channel 3^Output
	'}	
	{attribute 'pytmc' := '
		pv: TV2L0:GCC:01
		io: io
	'}
	TV2L0_GCC_01 : FB_MKS422;
	//HXR INSTALLATION SECTION 3
	{attribute 'TcLinkTo' := 	'.i_xOpnLS	:=	TIIB[EBD_E3_EL1004]^Channel 1^Input;
								 .i_xClsLS	:=	TIIB[EBD_E3_EL1004]^Channel 2^Input;
								 .q_xOPN_DO	:=	TIIB[EBD_E4_EL2004]^Channel 1^Output;
								 .q_xOPN_DO_2	:=	TIIB[EBD_E4_EL2004]^Channel 2^Output
	'}
	{attribute 'pytmc' := '
		pv: TV2L0:VGC:01
		io: io
	'}
	TV2L0_VGC_01 : FB_VGC_EBD;

	{attribute 'TcLinkTo' := 	'.i_iPRESS		:=	TIIB[QPC_E7_EL3064]^AI Standard Channel 2^Value;
								 .i_xSP_DI		:= 	TIIB[QPC_E8_EL1004]^Channel 2^Input;
								 .q_xHVEna_DO	:= 	TIIB[QPC_E9_EL2794]^Channel 2^Output
	'}	
	{attribute 'pytmc' := '
		pv: TV2L0:PIP:02
		io: io
	'}
	TV2L0_PIP_02 : FB_PIP_Gamma;
	
	{attribute 'TcLinkTo' := 	'.i_iPRESS_R	:=	TIIB[MKS_E18_EL3064]^AI Standard Channel 1^Value;
								 .q_xHV_DIS		:= 	TIIB[MKS_E20_EL2794]^Channel 1^Output
	'}	
	{attribute 'pytmc' := '
		pv: TV2L0:GFS:01
		io: io
	'}	
	TV2L0_GFS_01	:	FB_MKS422;
	
	{attribute 'TcLinkTo' := 	'.i_iPRESS_R	:=	TIIB[MKS_E5_EL3064]^AI Standard Channel 1^Value
	'}
	{attribute 'pytmc' := '
		pv: TV2L0:GPI:02
		io: io
	'}
	TV2L0_GPI_02 : FB_MKS317;

	{attribute 'TcLinkTo' := 	'.i_iPRESS_R	:=	TIIB[MKS_E4_EL3064]^AI Standard Channel 1^Value;
								 .q_xHV_DIS		:= 	TIIB[MKS_E6_EL2794]^Channel 1^Output
	'}	
	{attribute 'pytmc' := '
		pv: TV2L0:GCC:02
		io: io
	'}
	TV2L0_GCC_02 : FB_MKS422;

	{attribute 'TcLinkTo' := 	'.i_iPRESS		:=	TIIB[QPC_E7_EL3064]^AI Standard Channel 3^Value;
								 .i_xSP_DI		:= 	TIIB[QPC_E8_EL1004]^Channel 3^Input;
								 .q_xHVEna_DO	:= 	TIIB[QPC_E9_EL2794]^Channel 3^Output
	'}		
	{attribute 'pytmc' := '
		pv: TV2L0:PIP:03
		io: io
	'}
	TV2L0_PIP_03 : FB_PIP_Gamma;
	
	{attribute 'TcLinkTo' := 	'.i_xOpnLS	:=	TIIB[FEE_L0S2_EP1_EP2338-0002]^Channel 1^Input;
								 .i_xClsLS	:=	TIIB[FEE_L0S2_EP1_EP2338-0002]^Channel 2^Input;
								 .q_xOPN_DO	:=	TIIB[FEE_L0S2_EP1_EP2338-0002]^Channel 11^Output
	'}
	{attribute 'pytmc' := '
		pv: TV2L0:VGC:02
		io: io
	'}
	TV2L0_VGC_02 : FB_VGC;
	
(*SL1L0-POWER*) //HXR INSTALLATION SECTION 4
	{attribute 'TcLinkTo' := 	'.i_iPRESS_R	:=	TIIB[MKS_E9_EL3064]^AI Standard Channel 1^Value
	'}
	{attribute 'pytmc' := '
		pv: SL1L0:POWER:GPI:01
		io: io
	'}
	SL1L0_POWER_GPI_01 : FB_MKS317;

	{attribute 'TcLinkTo' := 	'.i_iPRESS_R	:=	TIIB[MKS_E8_EL3064]^AI Standard Channel 1^Value;
								 .q_xHV_DIS		:= 	TIIB[MKS_E10_EL2794]^Channel 1^Output
	'}	
	{attribute 'pytmc' := '
		pv: SL1L0:POWER:GCC:01
		io: io
	'}
	SL1L0_POWER_GCC_01 : FB_MKS422;

	{attribute 'TcLinkTo' := 	'.i_iPRESS		:=	TIIB[QPC_E21_EL3064]^AI Standard Channel 1^Value;
								 .i_xSP_DI		:= 	TIIB[QPC_E22_EL1004]^Channel 1^Input;
								 .q_xHVEna_DO	:= 	TIIB[QPC_E23_EL2794]^Channel 1^Output
	'}		
	{attribute 'pytmc' := '
		pv: SL1L0:POWER:PIN:01
		io: io
	'}
	SL1L0_POWER_PIN_01 : FB_PIP_Gamma;
	
(*AT2L0-SOLID*) //HXR INSTALLATION SECTION 6
	{attribute 'TcLinkTo' := 	'.i_iPRESS_R	:=	TIIB[MKS_E9_EL3064]^AI Standard Channel 2^Value
	'}
	{attribute 'pytmc' := '
		pv: AT2L0:SOLID:GPI:01
		io: io
	'}
	AT2L0_SOLID_GPI_01 : FB_MKS317;

	{attribute 'TcLinkTo' := 	'.i_iPRESS_R	:=	TIIB[MKS_E8_EL3064]^AI Standard Channel 3^Value;
								 .q_xHV_DIS		:= 	TIIB[MKS_E10_EL2794]^Channel 3^Output
	'}	
	{attribute 'pytmc' := '
		pv: AT2L0:SOLID:GCC:01
		io: io
	'}
	AT2L0_SOLID_GCC_01 : FB_MKS422;

	{attribute 'TcLinkTo' := 	'.i_iPRESS		:=	TIIB[QPC_E21_EL3064]^AI Standard Channel 2^Value;
								 .i_xSP_DI		:= 	TIIB[QPC_E22_EL1004]^Channel 2^Input;
								 .q_xHVEna_DO	:= 	TIIB[QPC_E23_EL2794]^Channel 2^Output
	'}	
	{attribute 'pytmc' := '
		pv: AT2L0:SOLID:PIN:01
		io: io
	'}
	AT2L0_SOLID_PIN_01 : FB_PIP_Gamma;
	
(*PC1L0-XTES*) //HXR INSTALLATION SECTION 7
	{attribute 'TcLinkTo' := 	'.i_xOpnLS	:=	TIIB[FEE_L0S8_EP1_EP2338-0002]^Channel 1^Input;
								 .i_xClsLS	:=	TIIB[FEE_L0S8_EP1_EP2338-0002]^Channel 2^Input;
								 .q_xOPN_DO	:=	TIIB[FEE_L0S8_EP1_EP2338-0002]^Channel 11^Output
	'}
	{attribute 'pytmc' := '
		pv: PC1L0:XTES:VGC:01
		io: io
	'}
	PC1L0_XTES_VGC_01 : FB_VGC;	
	
(*SP1L0-KMONO*)	
	{attribute 'TcLinkTo' := 	'.i_iPRESS_R	:=	TIIB[MKS_E12_EL3064]^AI Standard Channel 1^Value
	'}
	{attribute 'pytmc' := '
		pv: SP1L0:KMONO:GPI:01
		io: io
	'}
	SP1L0_KMONO_GPI_01 : FB_MKS317;

	{attribute 'TcLinkTo' := 	'.i_iPRESS_R	:=	TIIB[MKS_E11_EL3064]^AI Standard Channel 1^Value;
								 .q_xHV_DIS		:= 	TIIB[MKS_E13_EL2794]^Channel 1^Output
	'}	
	{attribute 'pytmc' := '
		pv: SP1L0:KMONO:GCC:01
		io: io
	'}
	SP1L0_KMONO_GCC_01 : FB_MKS422;

	{attribute 'TcLinkTo' := 	'.i_iPRESS		:=	TIIB[QPC_E11_EL3064]^AI Standard Channel 1^Value;
								 .i_xSP_DI		:= 	TIIB[QPC_E12_EL1004]^Channel 1^Input;
								 .q_xHVEna_DO	:= 	TIIB[QPC_E13_EL2794]^Channel 1^Output
	'}	
	{attribute 'pytmc' := '
		pv: SP1L0:KMONO:PIP:01
		io: io
	'}
	SP1L0_KMONO_PIP_01 : FB_PIP_Gamma;
	
(*PA1L0*)
	{attribute 'TcLinkTo' := 	'.i_iPRESS		:=	TIIB[QPC_E21_EL3064]^AI Standard Channel 3^Value;
								 .i_xSP_DI		:= 	TIIB[QPC_E22_EL1004]^Channel 3^Input;
								 .q_xHVEna_DO	:= 	TIIB[QPC_E23_EL2794]^Channel 3^Output
	'}
	{attribute 'pytmc' := '
		pv: PA1L0:PIN:01
		io: io
	'}
	PA1L0_PIN_01 : FB_PIP_Gamma; //PIN???	
	
	{attribute 'TcLinkTo' := 	'.q_xPress_OK		:= 	TIPC^plc_lfe_vac_fs^plc_lfe_vac_fs Instance^PlcTask Inputs^GVL_FS_Devices.PA1L0_VFS_01.i_xPress_OK;
								 .q_xVAC_FAULT_Reset:= 	TIPC^plc_lfe_vac_fs^plc_lfe_vac_fs Instance^PlcTask Inputs^GVL_FS_Devices.PA1L0_VFS_01.i_xResetFault;
								 .i_xTrigger		:=	TIPC^plc_lfe_vac_fs^plc_lfe_vac_fs Instance^PlcTask Outputs^GVL_FS_Devices.PA1L0_VFS_01.q_xTrigger;
								 .i_xVFS_Open		:=	TIPC^plc_lfe_vac_fs^plc_lfe_vac_fs Instance^PlcTask Outputs^GVL_FS_Devices.PA1L0_VFS_01.q_xVFS_Open;
								 .i_xVFS_Closed		:=	TIPC^plc_lfe_vac_fs^plc_lfe_vac_fs Instance^PlcTask Outputs^GVL_FS_Devices.PA1L0_VFS_01.q_xVFS_Closed;
								 .i_xVAC_FAULT_OK	:=	TIPC^plc_lfe_vac_fs^plc_lfe_vac_fs Instance^PlcTask Outputs^GVL_FS_Devices.PA1L0_VFS_01.q_xVAC_FAULT_OK
	'}
	{attribute 'pytmc' := '
		pv: PA1L0:VFS:01
		io: io
	'}	
	PA1L0_VFS_01	:	FB_VFS_Interface;
	
	{attribute 'TcLinkTo' := 	'.i_iPRESS_R	:=	TIIB[MKS_E15_EL3064]^AI Standard Channel 1^Value
	'}
	{attribute 'pytmc' := '
		pv: PA1L0:GPI:01
		io: io
	'}
	PA1L0_GPI_01 : FB_MKS317;

	{attribute 'TcLinkTo' := 	'.i_iPRESS_R	:=	TIIB[MKS_E14_EL3064]^AI Standard Channel 1^Value;
								 .q_xHV_DIS		:= 	TIIB[MKS_E16_EL2794]^Channel 1^Output
	'}	
	{attribute 'pytmc' := '
		pv: PA1L0:GCC:01
		io: io
	'}
	PA1L0_GCC_01 : FB_MKS422;
	
(*MR1L0-HOMS*) //HXR INSTALLATION SECTION 8
	{attribute 'TcLinkTo' := 	'.i_xOpnLS	:=	TIIB[FEE_L0S10_EP1_EP2338-0002]^Channel 1^Input;
								 .i_xClsLS	:=	TIIB[FEE_L0S10_EP1_EP2338-0002]^Channel 2^Input;
								 .q_xOPN_DO	:=	TIIB[FEE_L0S10_EP1_EP2338-0002]^Channel 11^Output
	'}
	{attribute 'pytmc' := '
		pv: MR1L0:HOMS:VGC:01
		io: io
	'}
	MR1L0_HOMS_VGC_01 : FB_VGC;	
	
	{attribute 'TcLinkTo' := 	'.i_iPRESS_R	:=	TIIB[MKS_E15_EL3064]^AI Standard Channel 2^Value
	'}
	{attribute 'pytmc' := '
		pv: MR1L0:HOMS:GPI:01
		io: io
	'}
	MR1L0_HOMS_GPI_01 : FB_MKS317;

	{attribute 'TcLinkTo' := 	'.i_iPRESS_R	:=	TIIB[MKS_E14_EL3064]^AI Standard Channel 3^Value;
								 .q_xHV_DIS		:= 	TIIB[MKS_E16_EL2794]^Channel 3^Output
	'}	
	{attribute 'pytmc' := '
		pv: MR1L0:HOMS:GCC:01
		io: io
	'}
	MR1L0_HOMS_GCC_01 : FB_MKS422;

	{attribute 'TcLinkTo' := 	'.i_iPRESS		:=	TIIB[QPC_E14_EL3064]^AI Standard Channel 4^Value;
								 .i_xSP_DI		:= 	TIIB[QPC_E15_EL1004]^Channel 4^Input;
								 .q_xHVEna_DO	:= 	TIIB[QPC_E16_EL2794]^Channel 4^Output
	'}	
	{attribute 'pytmc' := '
		pv: MR1L0:HOMS:PIP:01
		io: io
	'}
	MR1L0_HOMS_PIP_01 : FB_PIP_Gamma;
	
(*MR1L1-TXI*)
	{attribute 'TcLinkTo' := 	'.i_iPRESS_R	:=	TIIB[FEE_L0S14_EP2_EP3174-0002]^AI Standard Channel 1^Value
	'}
	{attribute 'pytmc' := '
		pv: MR1L1:TXI:GPI:01
		io: io
	'}
	MR1L1_TXI_GPI_01 : FB_MKS275;

	{attribute 'TcLinkTo' := 	'.i_iPRESS_R	:=	TIIB[FEE_L0S14_EP2_EP3174-0002]^AI Standard Channel 2^Value;
								 .q_xHV_DIS		:= 	TIIB[FEE_L0S14_EP3_EP2624-0002]^Channel 2^Output
	'}	
	{attribute 'pytmc' := '
		pv: MR1L1:TXI:GCC:01
		io: io
	'}
	MR1L1_TXI_GCC_01 : FB_MKS500_EP;

	{attribute 'TcLinkTo' := 	'.i_iPRESS		:=	TIIB[QPC_E14_EL3064]^AI Standard Channel 3^Value;
								 .i_xSP_DI		:= 	TIIB[QPC_E15_EL1004]^Channel 3^Input;
								 .q_xHVEna_DO	:= 	TIIB[QPC_E16_EL2794]^Channel 3^Output
	'}	
	{attribute 'pytmc' := '
		pv: MR1L1:TXI:PIP:01
		io: io
	'}
	MR1L1_TXI_PIP_01 : FB_PIP_Gamma;
	
(*BT2L0-PLEG*) //HXR INSTALLATION SECTION 9
	{attribute 'TcLinkTo' := 	'.i_xOpnLS	:=	TIIB[FEE_L0S14_EP1_EP2338-0002]^Channel 1^Input;
								 .i_xClsLS	:=	TIIB[FEE_L0S14_EP1_EP2338-0002]^Channel 2^Input;
								 .q_xOPN_DO	:=	TIIB[FEE_L0S14_EP1_EP2338-0002]^Channel 11^Output
	'}
	{attribute 'pytmc' := '
		pv: BT2L0:PLEG:VGC:01
		io: io
	'}
	BT2L0_PLEG_VGC_01 : FB_VGC;	
	
	{attribute 'TcLinkTo' := 	'.i_iPRESS_R	:=	TIIB[FEE_L0S14_EP2_EP3174-0002]^AI Standard Channel 3^Value
	'}
	{attribute 'pytmc' := '
		pv: BT2L0:PLEG:GPI:01
		io: io
	'}
	BT2L0_PLEG_GPI_01 : FB_MKS275;

	{attribute 'TcLinkTo' := 	'.i_iPRESS_R	:=	TIIB[FEE_L0S14_EP2_EP3174-0002]^AI Standard Channel 4^Value;
								 .q_xHV_DIS		:= 	TIIB[FEE_L0S14_EP3_EP2624-0002]^Channel 4^Output
	'}	
	{attribute 'pytmc' := '
		pv: BT2L0:PLEG:GCC:01
		io: io
	'}
	BT2L0_PLEG_GCC_01 : FB_MKS500_EP;

	{attribute 'TcLinkTo' := 	'.i_iPRESS		:=	TIIB[QPC_E11_EL3064]^AI Standard Channel 3^Value;
								 .i_xSP_DI		:= 	TIIB[QPC_E12_EL1004]^Channel 3^Input;
								 .q_xHVEna_DO	:= 	TIIB[QPC_E13_EL2794]^Channel 3^Output
	'}	
	{attribute 'pytmc' := '
		pv: BT2L0:PLEG:PIP:01
		io: io
	'}
	BT2L0_PLEG_PIP_01 : FB_PIP_Gamma;
	
(*MR2L0-HOMS*) //HXR INSTALLATION SECTION 10
	{attribute 'TcLinkTo' := 	'.i_xOpnLS	:=	TIIB[FEE_L0S18_EP1_EP2338-0002]^Channel 1^Input;
								 .i_xClsLS	:=	TIIB[FEE_L0S18_EP1_EP2338-0002]^Channel 2^Input;
								 .q_xOPN_DO	:=	TIIB[FEE_L0S18_EP1_EP2338-0002]^Channel 11^Output
	'}
	{attribute 'pytmc' := '
		pv: MR2L0:HOMS:VGC:01
		io: io
	'}
	MR2L0_HOMS_VGC_01 : FB_VGC;	
	
	{attribute 'TcLinkTo' := 	'.i_iPRESS_R	:=	TIIB[FEE_L0S18_EP2_EP3174-0002]^AI Standard Channel 1^Value
	'}
	{attribute 'pytmc' := '
		pv: MR2L0:HOMS:GPI:01
		io: io
	'}
	MR2L0_HOMS_GPI_01 : FB_MKS275;

	{attribute 'TcLinkTo' := 	'.i_iPRESS_R	:=	TIIB[FEE_L0S18_EP2_EP3174-0002]^AI Standard Channel 2^Value;
								 .q_xHV_DIS		:= 	TIIB[FEE_L0S18_EP3_EP2624-0002]^Channel 2^Output
	'}	
	{attribute 'pytmc' := '
		pv: MR2L0:HOMS:GCC:01
		io: io
	'}
	MR2L0_HOMS_GCC_01 : FB_MKS500_EP;

	{attribute 'TcLinkTo' := 	'.i_iPRESS		:=	TIIB[QPC_E11_EL3064]^AI Standard Channel 4^Value;
								 .i_xSP_DI		:= 	TIIB[QPC_E12_EL1004]^Channel 4^Input;
								 .q_xHVEna_DO	:= 	TIIB[QPC_E13_EL2794]^Channel 4^Output
	'}	
	{attribute 'pytmc' := '
		pv: MR2L0:HOMS:PIP:01
		io: io
	'}
	MR2L0_HOMS_PIP_01 : FB_PIP_Gamma;
	
	{attribute 'TcLinkTo' := 	'.i_xOpnLS	:=	TIIB[FEE_L0S19_EP1_EP2338-0002]^Channel 1^Input;
								 .i_xClsLS	:=	TIIB[FEE_L0S19_EP1_EP2338-0002]^Channel 2^Input;
								 .q_xOPN_DO	:=	TIIB[FEE_L0S19_EP1_EP2338-0002]^Channel 11^Output
	'}
	{attribute 'pytmc' := '
		pv: MR2L0:HOMS:VGC:02
		io: io
	'}
	MR2L0_HOMS_VGC_02 : FB_VGC;	
	
		
	{attribute 'TcLinkTo' := 	'.q_xPress_OK		:= 	TIPC^plc_lfe_vac_fs^plc_lfe_vac_fs Instance^PlcTask Inputs^GVL_FS_Devices.TV3L0_VFS_01.i_xPress_OK;
								 .q_xVAC_FAULT_Reset:= 	TIPC^plc_lfe_vac_fs^plc_lfe_vac_fs Instance^PlcTask Inputs^GVL_FS_Devices.TV3L0_VFS_01.i_xResetFault;
								 .i_xTrigger		:=	TIPC^plc_lfe_vac_fs^plc_lfe_vac_fs Instance^PlcTask Outputs^GVL_FS_Devices.TV3L0_VFS_01.q_xTrigger;
								 .i_xVFS_Open		:=	TIPC^plc_lfe_vac_fs^plc_lfe_vac_fs Instance^PlcTask Outputs^GVL_FS_Devices.TV3L0_VFS_01.q_xVFS_Open;
								 .i_xVFS_Closed		:=	TIPC^plc_lfe_vac_fs^plc_lfe_vac_fs Instance^PlcTask Outputs^GVL_FS_Devices.TV3L0_VFS_01.q_xVFS_Closed;
								 .i_xVAC_FAULT_OK	:=	TIPC^plc_lfe_vac_fs^plc_lfe_vac_fs Instance^PlcTask Outputs^GVL_FS_Devices.TV3L0_VFS_01.q_xVAC_FAULT_OK
	'}
	{attribute 'pytmc' := '
		pv: TV3L0:VFS:01
		io: io
	'}	
	TV3L0_VFS_01_Interface	:	FB_VFS_Interface;

(*TV1L1*)
	{attribute 'TcLinkTo' := 	'.i_xOpnLS	:=	TIIB[FEE_L0S18_EP1_EP2338-0002]^Channel 5^Input;
								 .i_xClsLS	:=	TIIB[FEE_L0S18_EP1_EP2338-0002]^Channel 6^Input;
								 .q_xOPN_DO	:=	TIIB[FEE_L0S18_EP1_EP2338-0002]^Channel 15^Output
	'}
	{attribute 'pytmc' := '
		pv: TV1L1:VGC:01
		io: io
	'}
	TV1L1_VGC_01 : FB_VGC;		

(*TV3L0*) //HXR INSTALLATION SECTION 11
(*
	{attribute 'pytmc' := '
		pv: TV3L0:VFS:01
		io: io
	'}
	TV3L0_VFS_01 : FB_VFS;
*)	
	{attribute 'TcLinkTo' := 	'.i_iPRESS		:=	TIIB[QPC_E14_EL3064]^AI Standard Channel 1^Value;
								 .i_xSP_DI		:= 	TIIB[QPC_E15_EL1004]^Channel 1^Input;
								 .q_xHVEna_DO	:= 	TIIB[QPC_E16_EL2794]^Channel 1^Output
	'}
	{attribute 'pytmc' := '
		pv: TV3L0:PIP:01
		io: io
	'}
	TV3L0_PIP_01 : FB_PIP_Gamma;
	
(*ST1L0-XTES*)
	{attribute 'TcLinkTo' := 	'.i_iPRESS_R	:=	TIIB[FEE_L0S21-2_EP1_EP3174-0002]^AI Standard Channel 1^Value
	'}
	{attribute 'pytmc' := '
		pv: ST1L0:XTES:GPI:01
		io: io
	'}
	ST1L0_XTES_GPI_01 : FB_MKS275;

	{attribute 'TcLinkTo' := 	'.i_iPRESS_R	:=	TIIB[FEE_L0S21-2_EP1_EP3174-0002]^AI Standard Channel 2^Value;
								 .q_xHV_DIS		:= 	TIIB[FEE_L0S21-2_EP2_EP2624-0002]^Channel 2^Output
	'}	
	{attribute 'pytmc' := '
		pv: ST1L0:XTES:GCC:01
		io: io
	'}
	ST1L0_XTES_GCC_01 : FB_MKS500_EP;

	{attribute 'TcLinkTo' := 	'.i_iPRESS		:=	TIIB[QPC_E14_EL3064]^AI Standard Channel 2^Value;
								 .i_xSP_DI		:= 	TIIB[QPC_E15_EL1004]^Channel 2^Input;
								 .q_xHVEna_DO	:= 	TIIB[QPC_E16_EL2794]^Channel 2^Output
	'}	
	{attribute 'pytmc' := '
		pv: ST1L0:XTES:PIP:01
		io: io
	'}
	ST1L0_XTES_PIP_01 : FB_PIP_Gamma;
	
(*PC2L1-L2SI*)
	{attribute 'TcLinkTo' := 	'.i_xOpnLS	:=	TIIB[FEE_L0S19_EP1_EP2338-0002]^Channel 5^Input;
								 .i_xClsLS	:=	TIIB[FEE_L0S19_EP1_EP2338-0002]^Channel 6^Input;
								 .q_xOPN_DO	:=	TIIB[FEE_L0S19_EP1_EP2338-0002]^Channel 15^Output
	'}
	{attribute 'pytmc' := '
		pv: PC2L1:L2SI:VGC:01
		io: io
	'}
	PC2L1_L2SI_VGC_01 : FB_VGC;

(*TV4L0*) // Hutch 1.1

	{attribute 'TcLinkTo' := 	'.i_iPRESS_R	:=	TIIB[H11_L0S2_EP2_EP3174-0002]^AI Standard Channel 1^Value
	'}
	{attribute 'pytmc' := '
		pv: TV4L0:GPI:01
		io: io
	'}
	TV4L0_GPI_01 : FB_MKS275;
	
	{attribute 'TcLinkTo' := 	'.i_iPRESS_R	:=	TIIB[H11_L0S2_EP2_EP3174-0002]^AI Standard Channel 2^Value;
								 .q_xHV_DIS		:= 	TIIB[H11_L0S2_EP3_EP2624-0002]^Channel 2^Output
	'}
	{attribute 'pytmc' := '
		pv: TV4L0:GCC:01
		io: io
	'}
	TV4L0_GCC_01 : FB_MKS500_EP;

	{attribute 'TcLinkTo' := 	'.i_iPRESS		:=	TIIB[QPC_E17_EL3064]^AI Standard Channel 1^Value;
								 .i_xSP_DI		:= 	TIIB[QPC_E18_EL1004]^Channel 1^Input;
								 .q_xHVEna_DO	:= 	TIIB[QPC_E19_EL2794]^Channel 1^Output
	'}	
	{attribute 'pytmc' := '
		pv: TV4L0:PIP:01
		io: io
	'}
	TV4L0_PIP_01 : FB_PIP_Gamma;
	
	{attribute 'TcLinkTo' := 	'.i_xOpnLS	:=	TIIB[H11_L0S2_EP1_EP2338-0002]^Channel 1^Input;
								 .i_xClsLS	:=	TIIB[H11_L0S2_EP1_EP2338-0002]^Channel 2^Input;
								 .q_xOPN_DO	:=	TIIB[H11_L0S2_EP1_EP2338-0002]^Channel 11^Output
	'}
	{attribute 'pytmc' := '
		pv: TV4L0:VGC:01
		io: io
	'}
	TV4L0_VGC_01 : FB_VGC;
	
	{attribute 'TcLinkTo' := 	'.i_iPRESS_R	:=	TIIB[H11_L0S9_EP1_EP3174-0002]^AI Standard Channel 1^Value
	'}
	{attribute 'pytmc' := '
		pv: TV4L0:GPI:02
		io: io
	'}
	TV4L0_GPI_02 : FB_MKS275;
	
	{attribute 'TcLinkTo' := 	'.i_iPRESS_R	:=	TIIB[H11_L0S9_EP1_EP3174-0002]^AI Standard Channel 2^Value;
								 .q_xHV_DIS		:= 	TIIB[H11_L0S9_EP2_EP2624-0002]^Channel 2^Output
	'}
	{attribute 'pytmc' := '
		pv: TV4L0:GCC:02
		io: io
	'}
	TV4L0_GCC_02 : FB_MKS500_EP;

	{attribute 'TcLinkTo' := 	'.i_iPRESS		:=	TIIB[QPC_E17_EL3064]^AI Standard Channel 2^Value;
								 .i_xSP_DI		:= 	TIIB[QPC_E18_EL1004]^Channel 2^Input;
								 .q_xHVEna_DO	:= 	TIIB[QPC_E19_EL2794]^Channel 2^Output
	'}		
	{attribute 'pytmc' := '
		pv: TV4L0:PIP:02
		io: io
	'}
	TV4L0_PIP_02 : FB_PIP_Gamma;

(*PA2L0*)
	{attribute 'TcLinkTo' := 	'.i_iPRESS		:=	TIIB[QPC_E21_EL3064]^AI Standard Channel 4^Value;
								 .i_xSP_DI		:= 	TIIB[QPC_E22_EL1004]^Channel 4^Input;
								 .q_xHVEna_DO	:= 	TIIB[QPC_E23_EL2794]^Channel 4^Output
	'}
	{attribute 'pytmc' := '
		pv: PA2L0:PIN:01
		io: io
	'}
	PA2L0_PIN_01 : FB_PIP_Gamma;


//Hutch 1.2
(*TV5L0*) 

	{attribute 'TcLinkTo' := 	'.i_iPRESS_R	:=	TIIB[H12_L0S1_EP1_EP3174-0002]^AI Standard Channel 1^Value
	'}
	{attribute 'pytmc' := '
		pv: TV5L0:GPI:01
		io: io
	'}
	TV5L0_GPI_01 : FB_MKS275;
	
	{attribute 'TcLinkTo' := 	'.i_iPRESS_R	:=	TIIB[H12_L0S1_EP1_EP3174-0002]^AI Standard Channel 2^Value;
								 .q_xHV_DIS		:= 	TIIB[H12_L0S1_EP2_EP2624-0002]^Channel 2^Output
	'}
	{attribute 'pytmc' := '
		pv: TV5L0:GCC:01
		io: io
	'}
	TV5L0_GCC_01 : FB_MKS500_EP;

	{attribute 'TcLinkTo' := 	'.i_iPRESS		:=	TIIB[QPC_E17_EL3064]^AI Standard Channel 3^Value;
								 .i_xSP_DI		:= 	TIIB[QPC_E18_EL1004]^Channel 3^Input;
								 .q_xHVEna_DO	:= 	TIIB[QPC_E19_EL2794]^Channel 3^Output
	'}		
	{attribute 'pytmc' := '
		pv: TV5L0:PIP:01
		io: io
	'}
	TV5L0_PIP_01 : FB_PIP_Gamma;
	
	{attribute 'TcLinkTo' := 	'.i_xOpnLS	:=	TIIB[H12_L0S3_EP1_EP2338-0002]^Channel 1^Input;
								 .i_xClsLS	:=	TIIB[H12_L0S3_EP1_EP2338-0002]^Channel 2^Input;
								 .q_xOPN_DO	:=	TIIB[H12_L0S3_EP1_EP2338-0002]^Channel 11^Output
	'}
	{attribute 'pytmc' := '
		pv: TV5L0:VGC:01
		io: io
	'}
	TV5L0_VGC_01 : FB_VGC;
	
	{attribute 'TcLinkTo' := 	'.i_iPRESS_R	:=	TIIB[H12_L0S3_EP2_EP3174-0002]^AI Standard Channel 1^Value
	'}
	{attribute 'pytmc' := '
		pv: TV5L0:GPI:02
		io: io
	'}
	TV5L0_GPI_02 : FB_MKS275;
	
	{attribute 'TcLinkTo' := 	'.i_iPRESS_R	:=	TIIB[H12_L0S3_EP2_EP3174-0002]^AI Standard Channel 2^Value;
								 .q_xHV_DIS		:= 	TIIB[H12_L0S3_EP3_EP2624-0002]^Channel 2^Output
	'}
	{attribute 'pytmc' := '
		pv: TV5L0:GCC:02
		io: io
	'}
	TV5L0_GCC_02 : FB_MKS500_EP;

	{attribute 'TcLinkTo' := 	'.i_iPRESS		:=	TIIB[QPC_E17_EL3064]^AI Standard Channel 4^Value;
								 .i_xSP_DI		:= 	TIIB[QPC_E18_EL1004]^Channel 4^Input;
								 .q_xHVEna_DO	:= 	TIIB[QPC_E19_EL2794]^Channel 4^Output
	'}		
	{attribute 'pytmc' := '
		pv: TV5L0:PIP:02
		io: io
	'}
	TV5L0_PIP_02 : FB_PIP_Gamma;

	{attribute 'TcLinkTo' := 	'.i_iPRESS_R	:=	TIIB[MKS_E18_EL3064]^AI Standard Channel 3^Value;
								 .q_xHV_DIS		:= 	TIIB[MKS_E20_EL2794]^Channel 2^Output
	'}	
	{attribute 'pytmc' := '
		pv: TV5L0:GFS:01
		io: io
	'}
	TV5L0_GFS_01 : FB_MKS422;

	{attribute 'TcLinkTo' := 	'.i_iPRESS_R	:=	TIIB[H12_L0S3_EP2_EP3174-0002]^AI Standard Channel 4^Value;
								 .q_xHV_DIS		:= 	TIIB[H12_L0S3_EP3_EP2624-0002]^Channel 4^Output
	'}
	{attribute 'pytmc' := '
		pv: TV5L0:GCC:03
		io: io
	'}
	TV5L0_GCC_03 : FB_MKS500_EP;

	{attribute 'TcLinkTo' := 	'.i_iPRESS		:=	TIIB[QPC_E4_EL3064]^AI Standard Channel 4^Value;
								 .i_xSP_DI		:= 	TIIB[QPC_E5_EL1004]^Channel 4^Input;
								 .q_xHVEna_DO	:= 	TIIB[QPC_E6_EL2794]^Channel 4^Output
	'}		
	{attribute 'pytmc' := '
		pv: TV5L0:PIP:03
		io: io
	'}
	TV5L0_PIP_03 : FB_PIP_Gamma;
	
(*TV6L0*)
	{attribute 'TcLinkTo' := 	'.i_xOpnLS	:=	TIIB[H12_L0S6_EP1_EP2338-0002]^Channel 1^Input;
								 .i_xClsLS	:=	TIIB[H12_L0S6_EP1_EP2338-0002]^Channel 2^Input;
								 .q_xOPN_DO	:=	TIIB[H12_L0S6_EP1_EP2338-0002]^Channel 11^Output
	'}
	{attribute 'pytmc' := '
		pv: TV6L0:VGC:01
		io: io
	'}
	TV6L0_VGC_01 : FB_VGC;


END_VAR

// ---- GVLs/GVL_Variables.TcGVL
//{attribute 'qualified_only'}
VAR_GLOBAL
	
	r_Accelerator_Setpoint	: REAL := 1E-12; (*unrealistic setpoint currently*)
	{attribute 'pytmc' := 'pv:VAC:OVRDON'}
	xSystemOverrideMode_EBD	: BOOL := FALSE; (* Global system override for the HXR Vacuum System EBD*)
	xSystemOverrideMode_FEE	: BOOL := FALSE; (* Global system override for the HXR Vacuum System FEE*)
	xSystemOverrideMode_H1_1_H1_2	: BOOL := FALSE; (* Global system override for the HXR Vacuum System Hutch1.1 and Hutch1.2*)
END_VAR

// ---- POUs/DIAGNOSTICS.TcPOU
PROGRAM DIAGNOSTICS
VAR
	//Change the PLC String Name to the actual PLC NAME
	sPLCName :STRING := 'PLC-LFE-VAC';
	//Link the sAMSNetID to the Etherat Master netID
	i_sAMSNetID AT %I*: AMSNETID;
	// DO NOT CHANGE
	sAMSNetID : STRING; //used for EPICS PV
	sLibVersion_LCLS_General : STRING;(* := stLibVersion_LCLS_General.sVersion*) ;
	fbEcatDiag:FB_EcatDiag;
	bAllSlaveStateGood : BOOL;
	bMasterStateGood :BOOL;
	iMasterState: WORD;
	sMasterState:STRING;
	nSlaveNumber : UINT;
	aiSlaveStates: ARRAY[1..256] OF BYTE;
	aEcSlaveInfo :  ARRAY[1..256] OF ST_EcDevice;
END_VAR

// Instaniating a call to the fbEcatDiag
fbEcatDiag(
	I_AMSNetId:=i_sAMSNetID , 
	i_xFirstPass:= _TaskInfo[1].FirstCycle, 
	q_xAllSlaveStatesGood=> bAllSlaveStateGood , 
	q_anTermStates=> aiSlaveStates, 
	q_xMasterStateGood=>bMasterStateGood , 
	q_nMasterState=> iMasterState, 
	q_sMasterState=> sMasterState , 
	q_astEcConfSlaveInfo=> aEcSlaveInfo , 
	q_nSlaves=> nSlaveNumber);

END_PROGRAM

// ---- POUs/MAIN.TcPOU
PROGRAM MAIN
VAR
	(*HXR Accelerator side PLC Interface*)
	{attribute 'TcLinkTo' :=	'TIIB[EBD_E5_EL1008]^Channel 1^Input;
	'}
	i_xUpstreamTreaty_PressOK	AT	%I*	:	BOOL;
	
//	{attribute 'TcLinkTo' :=	'TIIB[EBD_E8_EL2794]^Channel 1^Output;
//	'}
//	q_xUpstreamTreaty_PressOK	AT	%Q*	:	BOOL;
	
	(*HXR Gas Attenuator PLC Interface*)

	(*TXI PLC Interface*)

	(*XPP PLC Interface*)

	fbLogHandler : FB_LogHandler;
	
END_VAR

fbLogHandler();


// Run the Diagnostics PRG
DIAGNOSTICS();

(*HXR Accelerator side PLC Interface*)
//Update Accelerator Gauge Pressure Reading
//Accelerator_Upstream_Gauge.xPRESS_OK	:=	i_xUpstreamTreaty_PressOK;

IF(i_xUpstreamTreaty_PressOK) THEN
	Accelerator_Upstream_Gauge.xPRESS_OK 	:= TRUE;
	//Accelerator_Upstream_Gauge.eState 	:= gc_GaugeValidState;
	Accelerator_Upstream_Gauge.rPRESS	 	:= 5e-6; //torr
ELSE
	Accelerator_Upstream_Gauge.xPRESS_OK 	:= FALSE;
	//Accelerator_Upstream_Gauge.eState 	:= 1;
	Accelerator_Upstream_Gauge.rPRESS	 	:= 760;	//torr

END_IF

(*HXR Gas Attenuator PLC Interface*)

(*TXI PLC Interface*)

(*XPP PLC Interface*)


(*PIRANI Gauges*)

	TV1L0_GPI_01(PG=>);
	
	TV2L0_GPI_01(PG=>);
	
	TV2L0_GPI_02(PG=>);
	
	SL1L0_POWER_GPI_01(PG=>);
	
	AT2L0_SOLID_GPI_01(PG=>);
	
	SP1L0_KMONO_GPI_01(PG=>);
	
	PA1L0_GPI_01(PG=>);
	
	MR1L0_HOMS_GPI_01(PG=>);
	
	MR1L1_TXI_GPI_01(PG=>);
	
	BT2L0_PLEG_GPI_01(PG=>);
	
	MR2L0_HOMS_GPI_01(PG=>);
	
	ST1L0_XTES_GPI_01(PG=>);
	
	//H1.1 and H1.2
	TV4L0_GPI_01(PG=>);
	
	TV4L0_GPI_02(PG=>);

	TV5L0_GPI_01(PG=>);
	
	TV5L0_GPI_02(PG=>);
	
	
(*Cold Cathode Gauges*)
	
	TV1L0_GCC_01(PG:=TV1L0_GPI_01.PG,IG=>);
	
	TV2L0_GCC_01(PG:=TV2L0_GPI_01.PG, IG=>);
	
	TV2L0_GFS_01(PG:=TV2L0_GPI_02.PG,IG=>);
	
	TV2L0_GCC_02(PG:=TV2L0_GPI_02.PG,IG=>);
	
	SL1L0_POWER_GCC_01(PG:=SL1L0_POWER_GPI_01.PG,IG=>);
	
	AT2L0_SOLID_GCC_01(PG:=AT2L0_SOLID_GPI_01.PG,IG=>);
	
	SP1L0_KMONO_GCC_01(PG:=SP1L0_KMONO_GPI_01.PG,IG=>);
	
	PA1L0_GCC_01(PG:=PA1L0_GPI_01.PG,IG=>);
	
	MR1L0_HOMS_GCC_01(PG:=MR1L0_HOMS_GPI_01.PG,IG=>);
	
	MR1L1_TXI_GCC_01(PG:=MR1L1_TXI_GPI_01.PG,IG=>);
	
	BT2L0_PLEG_GCC_01(PG:=BT2L0_PLEG_GPI_01.PG,IG=>);
	
	MR2L0_HOMS_GCC_01(PG:=MR2L0_HOMS_GPI_01.PG,IG=>);
	
	ST1L0_XTES_GCC_01(PG:=ST1L0_XTES_GPI_01.PG,IG=>);

	//H1.1 and H1.2
	TV4L0_GCC_01(PG:=TV4L0_GPI_01.PG,IG=>);
	
	TV4L0_GCC_02(PG:=TV4L0_GPI_02.PG,IG=>);

	TV5L0_GCC_01(PG:=TV5L0_GPI_01.PG,IG=>);
	
	TV5L0_GCC_02(PG:=TV5L0_GPI_02.PG,IG=>);
	
	TV5L0_GFS_01(PG:=TV5L0_GPI_02.PG,IG=>);
	
	TV5L0_GCC_03(PG:=TV5L0_GPI_02.PG,IG=>);
	
	
	
(*Ion Pumps*)

	RTDSL0_PIP_01(i_stGauge:=TV1L0_GCC_01.IG, stPump=>);
	
	RTDSL0_PIP_02(i_stGauge:=TV1L0_GCC_01.IG, stPump=>);
	
	RTDSL0_PIP_03(i_stGauge:=TV1L0_GCC_01.IG, stPump=>);
	
	RTDSL0_PIP_04(i_stGauge:=TV1L0_GCC_01.IG, stPump=>);
	
	RTDSL0_PIP_05(i_stGauge:=TV1L0_GCC_01.IG, stPump=>);
	
	IM1L0_XTES_PIP_01(i_stGauge:=TV2L0_GCC_01.IG, stPump=>);
	
	TV2L0_PIP_01(i_stGauge:=TV2L0_GCC_01.IG, stPump=>);
	
	TV2L0_PIP_02(i_stGauge:=TV2L0_GCC_02.IG, stPump=>);
	
	TV2L0_PIP_03(i_stGauge:=TV2L0_GCC_02.IG, stPump=>);
	
	SL1L0_POWER_PIN_01(i_stGauge:=SL1L0_POWER_GPI_01.PG, stPump=>);
	
	AT2L0_SOLID_PIN_01(i_stGauge:=AT2L0_SOLID_GPI_01.PG, stPump=>);
	
	SP1L0_KMONO_PIP_01(i_stGauge:=SP1L0_KMONO_GPI_01.PG, stPump=>);
	
	PA1L0_PIN_01(i_stGauge:=SP1L0_KMONO_GPI_01.PG, stPump=>); //PIN???	Do I also need CC setpoint?
	
	MR1L0_HOMS_PIP_01(i_stGauge:=MR1L0_HOMS_GPI_01.PG, stPump=>);
	
	MR1L1_TXI_PIP_01(i_stGauge:=MR1L1_TXI_GPI_01.PG, stPump=>);
	
	BT2L0_PLEG_PIP_01(i_stGauge:=BT2L0_PLEG_GPI_01.PG, stPump=>);
	
	MR2L0_HOMS_PIP_01(i_stGauge:=MR2L0_HOMS_GPI_01.PG, stPump=>);
	
	TV3L0_PIP_01(i_stGauge:=ST1L0_XTES_GPI_01.PG, stPump=>);
	
	ST1L0_XTES_PIP_01(i_stGauge:=ST1L0_XTES_GPI_01.PG, stPump=>);
	
	
	//H1.1 and H1.2
	TV4L0_PIP_01(i_stGauge:=TV4L0_GPI_01.PG, stPump=>);
	
	TV4L0_PIP_02(i_stGauge:=TV4L0_GPI_01.PG, stPump=>);
	
	PA2L0_PIN_01(i_stGauge:=TV5L0_GPI_01.PG, stPump=>);
	
	TV5L0_PIP_01(i_stGauge:=TV5L0_GPI_01.PG, stPump=>);
	
	TV5L0_PIP_02(i_stGauge:=TV5L0_GPI_01.PG, stPump=>);
	
	TV5L0_PIP_03(i_stGauge:=TV5L0_GPI_01.PG, stPump=>);

(*Vacuum Gate Valve*)
	
	TV1L0_VGC_01(
	i_stUSG:= Accelerator_Upstream_Gauge, 
	i_stDSG:= RTDSL0_PIP_03.q_IG, 
	i_xDis_DPIlk:= FALSE , 
	i_xEPS_OK:= TRUE, 
	i_xPMPS_OK:= TRUE, 
	i_xExt_OK:= TRUE, 
	i_xOverrideMode:= xSystemOverrideMode_EBD, 
	i_xReset:= xReset_PMPS_FFO1, 
	iq_stValve=> , 
	xMPS_OK=> , 
	io_fbFFHWO:= g_FastFaultOutput1);
	
	IM1L0_XTES_VGC_01(
	i_stUSG:= RTDSL0_PIP_03.q_IG, 
	i_stDSG:= IM1L0_XTES_PIP_01.q_IG, 
	i_xDis_DPIlk:= FALSE , 
	i_xEPS_OK:= TRUE, 
	i_xPMPS_OK:= TRUE, 
	i_xExt_OK:= TRUE, 
	i_xOverrideMode:= xSystemOverrideMode_EBD, 
	i_xReset:= xReset_PMPS_FFO1, 
	iq_stValve=> , 
	xMPS_OK=> , 
	io_fbFFHWO:= g_FastFaultOutput1);

	TV2L0_VGC_01(
	i_stUSG:= TV2L0_PIP_01.q_IG, 
	i_stDSG:= TV2L0_PIP_02.q_IG, 
	i_xDis_DPIlk:= FALSE , 
	i_xEPS_OK:= TRUE, 
	i_xPMPS_OK:= TRUE, 
	i_xExt_OK:= TRUE, 
	i_xOverrideMode:= xSystemOverrideMode_EBD, 
	i_xReset:= xReset_PMPS_FFO1, 
	iq_stValve=> , 
	xMPS_OK=> , 
	io_fbFFHWO:= g_FastFaultOutput1);
	
	TV2L0_VGC_02(
	i_stUSG:= TV2L0_PIP_03.q_IG, 
	i_stDSG:= SL1L0_POWER_PIN_01.q_IG, 
	i_xDis_DPIlk:= FALSE , 
	i_xEPS_OK:= TRUE, 
	i_xPMPS_OK:= TRUE, 
	i_xExt_OK:= TRUE, 
	i_xOverrideMode:= xSystemOverrideMode_FEE, 
	i_xReset:= xReset_PMPS_FFO1, 
	iq_stValve=> , 
	xMPS_OK=> , 
	io_fbFFHWO:= g_FastFaultOutput1);
	
	PC1L0_XTES_VGC_01(
	i_stUSG:= AT2L0_SOLID_PIN_01.q_IG, 
	i_stDSG:= SP1L0_KMONO_PIP_01.q_IG, 
	i_xDis_DPIlk:= FALSE , 
	i_xEPS_OK:= TRUE, 
	i_xPMPS_OK:= TRUE, 
	i_xExt_OK:= TRUE, 
	i_xOverrideMode:= xSystemOverrideMode_FEE, 
	i_xReset:= xReset_PMPS_FFO1, 
	iq_stValve=> , 
	xMPS_OK=> , 
	io_fbFFHWO:= g_FastFaultOutput1);
	
//	PA1L0_VFS_01 : FB_VFS;

	MR1L0_HOMS_VGC_01(
	i_stUSG:= PA1L0_PIN_01.q_IG, 
	i_stDSG:= MR1L0_HOMS_PIP_01.q_IG, 
	i_xDis_DPIlk:= FALSE , 
	i_xEPS_OK:= TRUE, 
	i_xPMPS_OK:= TRUE, 
	i_xExt_OK:= TRUE, 
	i_xOverrideMode:= xSystemOverrideMode_FEE, 
	i_xReset:= xReset_PMPS_FFO1, 
	iq_stValve=> , 
	xMPS_OK=> , 
	io_fbFFHWO:= g_FastFaultOutput1);

	BT2L0_PLEG_VGC_01(
	i_stUSG:= MR1L0_HOMS_PIP_01.q_IG, 
	i_stDSG:= BT2L0_PLEG_PIP_01.q_IG, 
	i_xDis_DPIlk:= FALSE , 
	i_xEPS_OK:= TRUE, 
	i_xPMPS_OK:= TRUE, 
	i_xExt_OK:= TRUE, 
	i_xOverrideMode:= xSystemOverrideMode_FEE, 
	i_xReset:= xReset_PMPS_FFO1, 
	iq_stValve=> , 
	xMPS_OK=> , 
	io_fbFFHWO:= g_FastFaultOutput1);

	MR2L0_HOMS_VGC_01(
	i_stUSG:= BT2L0_PLEG_PIP_01.q_IG, 
	i_stDSG:= MR2L0_HOMS_PIP_01.q_IG, 
	i_xDis_DPIlk:= FALSE , 
	i_xEPS_OK:= TRUE, 
	i_xPMPS_OK:= TRUE, 
	i_xExt_OK:= TRUE, 
	i_xOverrideMode:= xSystemOverrideMode_FEE, 
	i_xReset:= xReset_PMPS_FFO1, 
	iq_stValve=> , 
	xMPS_OK=> , 
	io_fbFFHWO:= g_FastFaultOutput1);	
	
	MR2L0_HOMS_VGC_02(
	i_stUSG:= MR2L0_HOMS_PIP_01.q_IG, 
	i_stDSG:= ST1L0_XTES_PIP_01.q_IG, 
	i_xDis_DPIlk:= FALSE , 
	i_xEPS_OK:= TRUE, 
	i_xPMPS_OK:= TRUE, 
	i_xExt_OK:= TRUE, 
	i_xOverrideMode:= xSystemOverrideMode_FEE, 
	i_xReset:= xReset_PMPS_FFO1, 
	iq_stValve=> , 
	xMPS_OK=> , 
	io_fbFFHWO:= g_FastFaultOutput1);

	TV1L1_VGC_01(
	i_stUSG:= MR1L1_TXI_PIP_01.q_IG, 
	i_stDSG:= MR2L0_HOMS_PIP_01.q_IG, 
	i_xDis_DPIlk:= FALSE , 
	i_xEPS_OK:= TRUE, 
	i_xPMPS_OK:= TRUE, 
	i_xExt_OK:= TRUE, 
	i_xOverrideMode:= xSystemOverrideMode_FEE, 
	i_xReset:= xReset_PMPS_FFO1, 
	iq_stValve=> , 
	xMPS_OK=> , 
	io_fbFFHWO:= g_FastFaultOutput1);		

//	TV3L0_VFS_01 : FB_VFS;

//	PC2L1_L2SI_VGC_01 : FB_VGC;

	//H1.1
	TV4L0_VGC_01(
	i_stUSG:= TV4L0_GCC_01.IG, 
	i_stDSG:= TV4L0_GCC_02.IG, 
	i_xDis_DPIlk:= FALSE , 
	i_xEPS_OK:= TRUE, 
	i_xPMPS_OK:= TRUE, 
	i_xExt_OK:= TRUE, 
	i_xOverrideMode:= xSystemOverrideMode_H1_1_H1_2, 
	i_xReset:= xReset_PMPS_FFO2, 
	iq_stValve=> , 
	xMPS_OK=> , 
	io_fbFFHWO:= g_FastFaultOutput2);	
		
	TV5L0_VGC_01(
	i_stUSG:= TV5L0_GCC_01.IG, 
	i_stDSG:= TV5L0_GCC_02.IG, 
	i_xDis_DPIlk:= FALSE , 
	i_xEPS_OK:= TRUE, 
	i_xPMPS_OK:= TRUE, 
	i_xExt_OK:= TRUE, 
	i_xOverrideMode:= xSystemOverrideMode_H1_1_H1_2, 
	i_xReset:= xReset_PMPS_FFO2, 
	iq_stValve=> , 
	xMPS_OK=> , 
	io_fbFFHWO:= g_FastFaultOutput2);	
	
	TV6L0_VGC_01(
	i_stUSG:= TV5L0_GCC_03.IG, 
	i_stDSG:= XPP_Downstream_Vacuum, 
	i_xDis_DPIlk:= FALSE , 
	i_xEPS_OK:= TRUE, 
	i_xPMPS_OK:= TRUE, 
	i_xExt_OK:= TRUE, 
	i_xOverrideMode:= xSystemOverrideMode_H1_1_H1_2, 
	i_xReset:= xReset_PMPS_FFO2, 
	iq_stValve=> , 
	xMPS_OK=> , 
	io_fbFFHWO:= g_FastFaultOutput2);		

(*Vacuum Fast Shutter Valve*)

END_PROGRAM
